(* CODESYS project CtaAppWagoModBus1.0.0.2.library
   Description: Modbus Library der CTA
      Mit WAGO unterstüzung.
   Version: 1.0.0.2
   Title: CtaAppWagoModbus
   Author: SIS
   Company: CTA
   Placeholder: CtaAppWagoModbus
   DocFormat: reStructuredText
   CompiledLibraryCompatibilityVersion: CODESYS V3.5 SP16 Patch 3
   LanguageModelAttribute: qualified-access-only
   DefaultNamespace: CtaAppWagoModbus

Project tree, tasks and I/O mapping:
  libraries: WagoAppPlcModbus, 1.1.4.8 (WAGO); Standard, 3.5.18.0 (System); CtaVisSymbols, 1.0.0.0 (CTA); CtaSysConfig, 1.0.0.0 (CTA); CtaAppTime, 1.0.0.0 (CTA); CtaAppBmk, 1.0.0.0 (CTA); VisuSymbols, 4.5.0.0 (System); VisuDialogs, * (System); CtaSysBase, 1.0.0.0 (CTA); CtaAppModbus, 1.0.0.0 (CTA)
  40 Visualizations/
    SERVER/
      visualisation VIS_ModBusServer
      INFO/
        visualisation VIS_ModBusAccesInfo
      PARAMETER/
        SERIAL/
          visualisation VIS_ModBusParameter_SERIAL
        TCP/
          visualisation VIS_ModBusParameter_TCP
        UDP/
          visualisation VIS_ModBusParameter_UDP
        visualisation VIS_ModBus_PopUp
    CLIENT/
      SERIAL Client/
        SERIAL PORT/
          visualisation VIS_ModBusSerialPort
          PARAMETER/
            SERIAL/
              visualisation VIS_ModBusParameter_Serial_Port_Control
            visualisation VIS_ModBus_PopUp_Serial_Port_Control
        SERIAL Client/
          visualisation VIS_ModBusSerialNode
          POPUP/
            PARAMETER/
              visualisation VIS_ModBusParameter_SERIAL_Client
            visualisation VIS_ModBus_Serial_NodePopUp
          visualisation VIS_ModBusSerialNode_QUERRY
        visualisation VIS_SERIAL_LINE_HORIZONTAL
        visualisation VIS_SERIAL_LINE_VERTIKAL
        visualisation VIS_MODBUS_SERIAL_LINE
      NETWORK Client/
        visualisation VIS_ModBusNetworkPortTcp
        TCP/
          visualisation VIS_ModBusTcpNode_QUERRY
          visualisation VIS_ModBusTcpNode
          POPUP/
            PARAMETER/
              visualisation VIS_ModBusParameter_TCP_Client
            visualisation VIS_ModBus_Tcpl_NodePopUp
        UDP/
        visualisation VIS_MODBUS_TCP_LINE
        visualisation VIS_TCP_LINE_HORIZONTAL
        visualisation VIS_TCP_LINE_VERTIKAL
      visualisation VIS_MODBUS_LINE
    HELPER/
      visualisation VIS_IP_INPUT
      visualisation VIS_IP_PARAMETER
      visualisation VIS_IP_PARAMETER_QUERRY
      visualisation VIS_IP_PARAMETER_BASE
    BMK/
      visualisation Node_BMK
      visualisation Node_BMK_QUERY
    DIALOG/
      visualisation ModBusPopUp
  30 Program Organization Units/
    JOB/
      function block fbJOB [ST]: metCheckToUnlinkUnlock, metCheckQuerryAdr, metLock, proAllJobsDone, metSetQuerry, metSetWriteWord, metGetResponse, metQuerryAyWordToAyWord, metQuerryAyBoolToAyWord, metResponsAyWordToAyBool, metResponsAyWordToAyWord, metCallAfterResponse, FB_INIT, metAnalytic, metMaxQuantity, metResetMissingLastAdr, metResetMissingFirstAdr
    CLIENT/
      NETWORK Client/
        TCP/
          function block fbMbTcpClient [ST]: actKeepAlive, FB_INIT, metCheckOnError, metFc4ReadInputRegister, actFC04, metFc2ReadDiscretInput, actFC15, metFc1ReadCoils, metFc3ReadHoldingRegister, metFc15WriteMultipleCoil, metFc16WriteHoldingRegisters, actFC01, actFC03, actConfig, actFC02, actFC16, proNodeReference, actFC43, sMajorMinorRevision, sProductCode, sVendorName, proModBusOK, metFc5WriteCoil, metFc6WriteHoldingRegister, actFC05, actFC06, proModBusErrorText, proModBusEnabled, proITF_BMK, metITF_BMK, actDelay
          function block fbMbTcpPortControll [ST]: metMbTcpClient, metSyncClient
        UDP/
          function block fbMbUdpClient [ST]: actFC16, metCheckOnError, actFcUserQuerry, metFc4ReadInputRegister, actFC04, actFC02, metFc2ReadDiscretInput, FB_INIT, metFc1ReadCoils, metFc15WriteMultipleCoil, metFc16WriteHoldingRegisters, actFC01, actFC03, actFC15, metFc3ReadHoldingRegister, actConfig, actFC43, sProductCode, sVendorName, sMajorMinorRevision, proModBusOK, metFc5WriteCoil, metFc6WriteHoldingRegister, actFC05, actFC06, proModBusErrorText, proModBusEnabled, metITF_BMK, proITF_BMK, actDelay
      SERIAL Client/
        function block fbMbSerialClient [ST]: actFC16, actFC15, actFC03, actFC01, metFc16WriteHoldingRegisters, metFc15WriteMultipleCoil, metFc3ReadHoldingRegister, metFc1ReadCoils, metCheckOnError, metFc2ReadDiscretInput, actFC02, actFC04, metFc4ReadInputRegister, FB_INIT, actConfig, proNodeReference, actFC43, sMajorMinorRevision, sProductCode, sVendorName, proModBusOK, actFC05, actFC06, metFc5WriteCoil, metFc6WriteHoldingRegister, proModBusErrorText, proModBusEnabled, metITF_BMK, proITF_BMK, actDelay
        function block fbMbSerialPortControll [ST]: metSyncClient, metMbSerialClient, actConfig
    SERVER/
      function block fbModBusServer [ST]: actConfig, actModBusServerTcp, actModBusServerUdp, actModBusServerSerial, metGetCoil, metSetDiscretInput, metGetHoldingRegister, metSetInputRegister, metAddSerialControll, metAddTcpControll, metAddUdpControll, metSetHoldingRegister, metSetCoil
      ACCES CONTROLL/
        function block fbAccesControll [ST]: beforeAccess, afterAccess, ALLOWBOOL
    CONVERTER/
      function fcWordBitToByte [ST]
      function fcCheckIp [ST]
      function fcSetInitialIPString [ST]
  00000000-0000-0000-0000-000000000000|D:\CoDeSys\LibrariesV3\trunk\Intern\CAA\CAA Template\3.4.0.0 draft\Placeholder.xml
  00000000-0000-0000-0000-000000000000|D:\CoDeSys\LibrariesV3\trunk\Intern\CAA\CAA Template\3.2.0.3 draft\Prefix.pdf
  00000000-0000-0000-0000-000000000000|D:\CoDeSys\LibrariesV3\trunk\Intern\CAA\CAA Template\3.5.2.0 draft\Placeholder.xml
  20 Structs/
    SERVER/
      PARAMETER/
        data type scModBusServerParameter
        TCP/
          data type scTcp
        UDP/
          data type scUdp
        SERIAL/
          data type scSerial
    CLIENT/
      SERIAL/
        data type scSerialPortParameter
        data type scSerialClientParameter
      NETWORK/
        data type scUdpClientParameter
        data type scTcpClientParameter
  50 Images/
  10 Documenation/
    global variables VersionHistory
    global variables readMe
  21 Interface/
    RTU/
      interface ITF_MbPortControllSerial: metMbSerialClient, metSyncClient
      interface ITF_SERIAL_NODE: proNodeReference
    ALL/
      interface ITF_MbClient: metFc16WriteHoldingRegisters, metFc15WriteMultipleCoil, metFc4ReadInputRegister, metFc3ReadHoldingRegister, metFc2ReadDiscretInput, metFc1ReadCoils, sProductCode, sVendorName, sMajorMinorRevision, proModBusOK, metFc5WriteCoil, metFc6WriteHoldingRegister, proModBusErrorText, proModBusEnabled, proITF_BMK, metITF_BMK
    NETWORK/
      interface ITF_TCP_NODE: proNodeReference
      interface ITF_UDP_NODE: proNodeReference
      interface ITF_MbPortControllTcp: metMbTcpClient, metSyncClient
    SERVER/
      interface ITF_SERVER: metAddSerialControll, metAddTcpControll, metAddUdpControll
  11 Library Parameter/
    global variables Parameter
  12 Konstanten/
  60 Textlisten/
    SERIAL/
      text list txtPhysikalLayer
      text list txtParity
      text list txtHandshake
      text list txtStopBits
  13 Globale Variablen/
    global variables GVL_CtaModBus
  text list GlobalTextList
*)

// 20 Structs/SERVER/PARAMETER/scModBusServerParameter
TYPE scModBusServerParameter :
    STRUCT
        scSerial    :   scSerial;
        scTcp       :   scTcp;
        scUdp       :   scUdp;
    END_STRUCT
END_TYPE

// 20 Structs/SERVER/PARAMETER/SERIAL/scSerial
TYPE scSerial :
    STRUCT
        fbxEnable           :   CtaSysConfig.fbBOOL;           // Serial Server Enable
        fbbyUnitId          :   CtaSysConfig.fbBYTE;           // Serial Server Id
        fbudiBaudrate       :   CtaSysConfig.fbUDINT;          // Serial Server Baudrate
        fbusiDataBits       :   CtaSysConfig.fbUSINT;          // Serial Server Databits 5..8
        fbiParity           :   CtaSysConfig.fbINT;            // WagoTypesCom.eTTYParity
        fbiStopBits         :   CtaSysConfig.fbINT;            // WagoTypesCom.eTTYStopBits
        fbiHandshake        :   CtaSysConfig.fbINT;            // WagoTypesCom.eTTYHandshake
        fbiPhysikal         :   CtaSysConfig.fbINT;            // WagoTypesCom.eTTYPhysicalLayer
        fbxRtuOrAscii       :   CtaSysConfig.fbBOOL;           // RTU = FALSE , ASCII = TRUE
        fbxEnableWatchDog   :   CtaSysConfig.fbBOOL;           // WatchDog Enable
        fbtWatchDog         :   CtaSysConfig.fbTIME;           // WatchDog Time
    END_STRUCT
END_TYPE

// 20 Structs/SERVER/PARAMETER/TCP/scTcp
TYPE scTcp :
    STRUCT
        fbxEnable           :   CtaSysConfig.fbBOOL;           // Tcp Server Enable    
        fbbyUnitId          :   CtaSysConfig.fbBYTE;           // Tcp Server Id
        fbwPort             :   CtaSysConfig.fbWORD;           // Tcp Server Port
        fbxKeepAlive        :   CtaSysConfig.fbBOOL;           // Tcp Server Keep Alive 
        fbtMaxIdleTime      :   CtaSysConfig.fbTIME;           // Tcp Server Max Offline Time
        fbtIntervall        :   CtaSysConfig.fbTIME;           // Tcp Server Intervall Time
        fbudiProbes         :   CtaSysConfig.fbUDINT;          // Tcp Server Retrys before give up 
        fbxEnableWatchDog   :   CtaSysConfig.fbBOOL;           // WatchDog Enable
        fbtWatchDog         :   CtaSysConfig.fbTIME;           // WatchDog Time
    END_STRUCT
END_TYPE

// 20 Structs/SERVER/PARAMETER/UDP/scUdp
TYPE scUdp :
    STRUCT
        fbxEnable       :   CtaSysConfig.fbBOOL;           // Udp Server Enable    
        fbbyUnitId      :   CtaSysConfig.fbBYTE;           // Udp Server Id
        fbwPort         :   CtaSysConfig.fbWORD;           // Udp Server Port  
        fbxEnableWatchDog   :   CtaSysConfig.fbBOOL;           // WatchDog Enable      
        fbtWatchDog     :   CtaSysConfig.fbTIME;           // WatchDog Time
    END_STRUCT
END_TYPE

// 20 Structs/CLIENT/NETWORK/scUdpClientParameter
TYPE scUdpClientParameter :
    STRUCT
        fbxEnable           :   CtaSysConfig.fbBOOL;           // Serial Server Enable        
        fbbyUnitId          :   CtaSysConfig.fbBYTE;           // Serial Server Id  
        fbstIp              :   CtaSysConfig.fbSTRING40;       // IP Adresse    
        fbwPort             :   CtaSysConfig.fbWORD;           // Port Nr          
        fbtTimeOut          :   CtaSysConfig.fbTIME;           // Timeout Time
        fbtScanRate         :   CtaSysConfig.fbTIME;           // Scan Rate Time
		fbtDelayRead		:	CtaSysConfig.fbTIME;		   // Read Delay
		fbtDelayWrite		:	CtaSysConfig.fbTIME;		   // Write Delay
    END_STRUCT
END_TYPE

// 20 Structs/CLIENT/SERIAL/scSerialPortParameter
TYPE scSerialPortParameter :
    STRUCT 
        fbudiBaudrate       :   CtaSysConfig.fbUDINT;          // Serial Server Baudrate
        fbusiDataBits       :   CtaSysConfig.fbUSINT;          // Serial Server Databits 5..8
        fbiParity           :   CtaSysConfig.fbINT;            // WagoTypesCom.eTTYParity
        fbiStopBits         :   CtaSysConfig.fbINT;            // WagoTypesCom.eTTYStopBits
        fbiHandshake        :   CtaSysConfig.fbINT;            // WagoTypesCom.eTTYHandshake
        fbiPhysikal         :   CtaSysConfig.fbINT;            // WagoTypesCom.eTTYPhysicalLayer
        fbxRtuOrAscii       :   CtaSysConfig.fbBOOL;           // RTU = FALSE , ASCII = TRUE
    END_STRUCT
END_TYPE

// 20 Structs/CLIENT/SERIAL/scSerialClientParameter
TYPE scSerialClientParameter :
    STRUCT
        fbxEnable           :   CtaSysConfig.fbBOOL;           // Serial Server Enable        
        fbbyUnitId          :   CtaSysConfig.fbBYTE;           // Serial Server Id        
        fbtTimeOut          :   CtaSysConfig.fbTIME;           // Timeout Time
        fbtScanRate         :   CtaSysConfig.fbTIME;           // Scan Rate Time
		fbtDelayRead		:	CtaSysConfig.fbTIME;		   // Read Delay
		fbtDelayWrite		:	CtaSysConfig.fbTIME;		   // Write Delay
    END_STRUCT
END_TYPE

// 20 Structs/CLIENT/NETWORK/scTcpClientParameter
TYPE scTcpClientParameter :
    STRUCT
        fbxEnable           :   CtaSysConfig.fbBOOL;           // Serial Server Enable       
        fbbyUnitId          :   CtaSysConfig.fbBYTE;           // Serial Server Id  
        fbstIp              :   CtaSysConfig.fbSTRING40;       // IP Adresse    
        fbwPort             :   CtaSysConfig.fbWORD;           // Port Nr          
        fbtTimeOut          :   CtaSysConfig.fbTIME;           // Timeout Time
        fbtScanRate         :   CtaSysConfig.fbTIME;           // Scan Rate Time
        fbxKeepAlive        :   CtaSysConfig.fbBOOL;           // Tcp Server Keep Alive 
        fbtMaxIdleTime      :   CtaSysConfig.fbTIME;           // Tcp Server Max Offline Time
        fbtIntervall        :   CtaSysConfig.fbTIME;           // Tcp Server Intervall Time
        fbudiProbes         :   CtaSysConfig.fbUDINT;          // Tcp Server Retrys before give up     
		fbtDelayRead		:	CtaSysConfig.fbTIME;		   // Read Delay
		fbtDelayWrite		:	CtaSysConfig.fbTIME;		   // Write Delay   
    END_STRUCT
END_TYPE

// 10 Documenation/VersionHistory
(* 

.. image:: ../../Images/CTA_Logo.jpg
   :align: right
   :width: 15% 

**Vorlage**   


============ =========== =========== ============================================
**Date**     **Version** **Author**  **Change**
------------ ----------- ----------- --------------------------------------------
04.03.2021   0.0.0.0     SIS         Vorlage erstellt

============ =========== =========== ============================================


*)
VAR_GLOBAL
    stInfo : STRING:= '0.0.0.0, Vorlage, CTA';
END_VAR

// 10 Documenation/readMe
(*

**ReadMe**
 
|	**Empfehlung**
|
|	Dokumentrieren Sie die Library für eine nachhaltige Entwicklung
|     
| *Beispiel* 
|
| Dies ist die Vorlage Library der CTA. Erstellen Sie ihre Library anhand dieser Vorlage.
*)

VAR_GLOBAL
    xReadMeDone              :   BOOL;
END_VAR

// 13 Globale Variablen/GVL_CtaModBus
{attribute 'qualified_only'}
VAR_GLOBAL   
    // {attribute 'hide'}
    byCountServer           : BYTE;     
    // {attribute 'hide'}     
    fbDeviceName            : WagoAppPlcModbus.FbIdentifyBaseObject:= ( _sVendorName            := Parameter.sVendorName,          
                                                                        _sProductCode           := Parameter.sProductCode,         
                                                                        _sMajorMinorRevision    := Parameter.sMajorMinorRevision);          
                                                      
END_VAR

// 11 Library Parameter/Parameter
{attribute 'qualified_only'}
VAR_GLOBAL CONSTANT
    sVendorName                 :   STRING(WagoAppPlcModbus.Parameter.MAX_IDENTIFICATION_MEMBER_LENGTH) := 'CTA AG';   
    sProductCode                :   STRING(WagoAppPlcModbus.Parameter.MAX_IDENTIFICATION_MEMBER_LENGTH) := 'CTA ModBus Device';
    sMajorMinorRevision         :   STRING(WagoAppPlcModbus.Parameter.MAX_IDENTIFICATION_MEMBER_LENGTH) := '1.0';    
    wQuantityReadTcpWord        :   WORD    :=  123;
    wQuantityReadTcpBool        :   WORD    := 1968;
    wQuantityReadSerialWord     :   WORD    :=  123;
    wQuantityReadSerialBool     :   WORD    := 1968;     
    wQuantityWriteTcpWord       :   WORD    :=  123;
    wQuantityWriteTcpBool       :   WORD    := 1968;
    wQuantityWriteSerialWord    :   WORD    :=   68;
    wQuantityWriteSerialBool    :   WORD    :=  123; 
END_VAR

// 30 Program Organization Units/CLIENT/SERIAL Client/fbMbSerialClient
FUNCTION_BLOCK fbMbSerialClient EXTENDS CtaSysBase.fbBASE IMPLEMENTS ITF_MbClient, ITF_SERIAL_NODE
VAR_INPUT
    ITF_MbPortControll          : ITF_MbPortControllSerial;   
END_VAR
VAR_OUTPUT
    xError                      : BOOL;
END_VAR
VAR
	ITF_BMK 					: CtaAppBmk.ITF_BMK;	
    xComAktive                  : BOOL;
    xDisabled                   : BOOL;
    byUnitId                    : BYTE;
    ITF_MbPortControllQuerry    : ITF_MbPortControllSerial; 
    xPortControllError          : BOOL;
    uiCountErrors               : UINT;    
    usiState                    : USINT := 1;
    fbTIMEFcs                   : CtaAppTime.fbTimeMeasurement;
    ltMessungFcs                : LTIME; 
    bIdOfCall                   : BYTE;
    TON_ScanRate                : TON;
    tonDelayRead				: Standard.TON;
	tonDelayWrite				: Standard.TON;
	xTrigDelayRead				: BOOL;
	xTrigDelayWrite				: BOOL; 
    xAllJobsDone                : BOOL;

    xErrorMbClientSerial        : BOOL;
    uiIdMbClientSerial          : UINT;
    
    
    (* FC1 *)
    fbJobFc1                    : fbJOB;
    xTrigFc1                    : BOOL;
    fbTIMEFc1                   : CtaAppTime.fbTimeMeasurement;
    ltMessungFc1                : LTIME;      
    (* FC2 *)
    fbJobFc2                    : fbJOB;
    xTrigFc2                    : BOOL; 
    fbTIMEFc2                   : CtaAppTime.fbTimeMeasurement;
    ltMessungFc2                : LTIME;      
    (* FC3 *)
    fbJobFc3                    : fbJOB;
    xTrigFc3                    : BOOL;      
    fbTIMEFc3                   : CtaAppTime.fbTimeMeasurement;
    ltMessungFc3                : LTIME;          
    (* FC4 *)
    fbJobFc4                    : fbJOB;
    xTrigFc4                    : BOOL;      
    fbTIMEFc4                   : CtaAppTime.fbTimeMeasurement;
    ltMessungFc4                : LTIME;      
    (* FC5 *)
    fbJobFc5                    : fbJOB;
    xTrigFc5                    : BOOL;      
    fbTIMEFc5                   : CtaAppTime.fbTimeMeasurement;
    ltMessungFc5                : LTIME;      
    (* FC6 *)
    fbJobFc6                    : fbJOB;
    xTrigFc6                    : BOOL;      
    fbTIMEFc6                   : CtaAppTime.fbTimeMeasurement;
    ltMessungFc6                : LTIME;      
    (* FC15 *)
    fbJobFc15                   : fbJOB;
    xTrigFc15                   : BOOL;   
    fbTIMEFc15                  : CtaAppTime.fbTimeMeasurement;
    ltMessungFc15               : LTIME;     
    (* FC16 *)   
    fbJobFc16                   : fbJOB;             
    xTrigFc16                   : BOOL;
    fbTIMEFc16                  : CtaAppTime.fbTimeMeasurement;
    ltMessungFc16               : LTIME;       
    (* FC43 *)   
    fbIdentifyObject			: WagoAppPlcModbus.FbIdentifyBaseObject;
	fbIdentifyMember3			: WagoAppPlcModbus.FbIdentifyMember_STRING(fbIdentifyObject,3);
	fbIdentifyMember4			: WagoAppPlcModbus.FbIdentifyMember_STRING(fbIdentifyObject,4);
	utIdentifyQuerry			: WagoAppPlcModbus.typMbQuery;
	utIdentifyResponse			: WagoAppPlcModbus.typMbResponse;           
    xTrigFc43                   : BOOL;
	xActiveFc43					: BOOL;
	xDoneFc43					: BOOL;
	tTimeOutFc43				: TIME;
    fbTIMEFc43                  : CtaAppTime.fbTimeMeasurement;
    ltMessungFc43               : LTIME;       	
    (* Parameter *)
    fbConfigFile                : CtaSysConfig.fbConfigFile;
    scParameter                 : scSerialClientParameter;    
END_VAR

(* Config File *)
actConfig();
(* Unit ID *)
byUnitId := scParameter.fbbyUnitId.byValue;
(* Is Enabled *)
IF scParameter.fbxEnable.xValue THEN
    (* Port Sync *)
    IF __QUERYINTERFACE(ITF_MbPortControll,ITF_MbPortControllQuerry) THEN
        xPortControllError := FALSE;  
        IF ITF_MbPortControllQuerry.metSyncClient(xAllJobsDone,bIdOfCall,THIS^) THEN
			(* Delay *)
			actDelay();
            (* FC1 *)
            actFC01();
            (* FC2 *)
            actFC02();
            (* FC3 *)
            actFC03();
            (* FC4 *)
            actFC04();
            (* FC5 *)
            actFC05();
            (* FC6 *)
            actFC06();
            (* FC15 *)
            actFC15();
            (* FC16 *)
            actFC16(); 
            (* FC43 *)
            actFC43(); 			
        END_IF;
    ELSE
        xPortControllError := TRUE;    
    END_IF;
    IF usiState >= 10 OR usiState = 0 THEN
        (* Check if all Jobs Done *)
        IF  fbJobFc1.xAllJobsDone  AND
            fbJobFc2.xAllJobsDone  AND
            fbJobFc3.xAllJobsDone  AND
            fbJobFc4.xAllJobsDone  AND
            fbJobFc5.xAllJobsDone  AND
            fbJobFc6.xAllJobsDone  AND			
            fbJobFc15.xAllJobsDone AND
            fbJobFc16.xAllJobsDone THEN
            (*Scan Rate *)
            TON_ScanRate(IN := NOT TON_ScanRate.Q,
                         PT := scParameter.fbtScanRate.tValue);
            xAllJobsDone := TRUE;             
            IF TON_ScanRate.Q THEN
                fbJobFc1.proAllJobsDone  := FALSE;
                fbJobFc2.proAllJobsDone  := FALSE;   
                fbJobFc3.proAllJobsDone  := FALSE;  
                fbJobFc4.proAllJobsDone  := FALSE;   
                fbJobFc5.proAllJobsDone  := FALSE;  
                fbJobFc6.proAllJobsDone  := FALSE; 	
                fbJobFc15.proAllJobsDone := FALSE;  
                fbJobFc16.proAllJobsDone := FALSE; 
                xAllJobsDone             := FALSE;    
                usiState := 1;
                (* Timer stopp *) 
                ltMessungFcs := fbTIMEFcs.stop();             
                (* Timer start *) 
                fbTIMEFcs.Start();      
            END_IF;        
        ELSE    
            usiState := 1;
        END_IF;   
    END_IF;
    
    xComAktive := fbJobFc1.wCountJobs  <> 0 OR 
                  fbJobFc2.wCountJobs  <> 0 OR
                  fbJobFc3.wCountJobs  <> 0 OR 
                  fbJobFc4.wCountJobs  <> 0 OR 
                  fbJobFc5.wCountJobs  <> 0 OR 
                  fbJobFc6.wCountJobs  <> 0 OR 				  
                  fbJobFc15.wCountJobs <> 0 OR
                  fbJobFc16.wCountJobs <> 0 ;  
                  
    (* Get Errors *)
    xError :=  fbJobFc1.eError <> WagoAppPlcModbus.eErrorModbus.OK OR 
               fbJobFc2.eError <> WagoAppPlcModbus.eErrorModbus.OK OR 
               fbJobFc3.eError <> WagoAppPlcModbus.eErrorModbus.OK OR 
               fbJobFc4.eError <> WagoAppPlcModbus.eErrorModbus.OK OR 
               fbJobFc5.eError <> WagoAppPlcModbus.eErrorModbus.OK OR 
               fbJobFc6.eError <> WagoAppPlcModbus.eErrorModbus.OK OR 			   
              fbJobFc15.eError <> WagoAppPlcModbus.eErrorModbus.OK OR 
              fbJobFc16.eError <> WagoAppPlcModbus.eErrorModbus.OK OR
              fbConfigFile.xError                                  OR
              xPortControllError;   
              
    IF NOT xError THEN
       uiCountErrors := 0;
    END_IF;
ELSE
    (* Reset States *)
    (* Port Sync *)
    IF __QUERYINTERFACE(ITF_MbPortControll,ITF_MbPortControllQuerry) THEN
        xPortControllError := FALSE;  
        xAllJobsDone       := FALSE;
        usiState           := 0;
        xError             := FALSE;
        xComAktive         := FALSE;
        xDisabled          := TRUE;
		xDoneFc43		   := FALSE;
        ITF_MbPortControllQuerry.metSyncClient(xDisabled,bIdOfCall,THIS^);
    END_IF; 
END_IF;

ACTION actFC16:
(* Trig FC16 *)
IF fbJobFc16.xIsLinked AND fbJobFc16.xIsQuerryReady AND NOT fbJobFc16.xIsLocked AND NOT fbJobFc16.xAllJobsDone AND tonDelayWrite.Q THEN
    fbJobFc16.metLock();
    xTrigFc16       := TRUE;
    fbTIMEFc16.Start();
ELSIF usiState = 8 AND (NOT fbJobFc16.xIsLinked OR fbJobFc16.xAllJobsDone) THEN
    usiState                    := usiState + 1; 
    fbJobFc16.proAllJobsDone    := TRUE;   
END_IF
(* Send Querry *)
IF usiState = 8 AND xTrigFc16 THEN
	xTrigDelayWrite := FALSE;
    ITF_MbPortControllQuerry.metMbSerialClient( tTimeOut    := scParameter.fbtTimeOut.tValue, 
                                                utQuery     := fbJobFc16.utQuery,
                                                xTrigger    := xTrigFc16,
                                                utResponse  := fbJobFc16.utResponse,
                                                xError      => xErrorMbClientSerial,
                                                uiID        => uiIdMbClientSerial);      
END_IF;
(* Get Response *) 
IF usiState = 8 AND NOT xTrigFc16 AND fbJobFc16.xIsLocked AND NOT fbJobFc16.xJobDone THEN    
    usiState            := usiState + 1;
    ltMessungFc16       := fbTIMEFc16.Stop();
    metCheckOnError(xErrorMbClientSerial);
    fbJobFc16.metCallAfterResponse(xErrorMbClientSerial,uiIdMbClientSerial);
END_IF;
END_ACTION

ACTION actFC15:
(* Trig FC15 *)
IF fbJobFc15.xIsLinked AND fbJobFc15.xIsQuerryReady AND NOT fbJobFc15.xIsLocked AND NOT fbJobFc15.xAllJobsDone AND tonDelayWrite.Q THEN
    fbJobFc15.metLock();
    xTrigFc15       := TRUE;
    fbTIMEFc15.Start();
ELSIF usiState = 7 AND (NOT fbJobFc15.xIsLinked OR fbJobFc15.xAllJobsDone) THEN
    usiState                    := usiState + 1; 
    fbJobFc15.proAllJobsDone    := TRUE;   
END_IF
(* Send Querry *)
IF usiState = 7 AND xTrigFc15 THEN
	xTrigDelayWrite := FALSE;
    ITF_MbPortControllQuerry.metMbSerialClient( tTimeOut    := scParameter.fbtTimeOut.tValue, 
                                                utQuery     := fbJobFc15.utQuery,
                                                xTrigger    := xTrigFc15,
                                                utResponse  := fbJobFc15.utResponse,
                                                xError      => xErrorMbClientSerial,
                                                uiID        => uiIdMbClientSerial); 
END_IF;
(* Get Response *) 
IF usiState = 7 AND NOT xTrigFc15 AND fbJobFc15.xIsLocked AND NOT fbJobFc15.xJobDone  THEN 
    usiState            := usiState + 1;
    ltMessungFc15       := fbTIMEFc15.Stop();
    metCheckOnError(xErrorMbClientSerial);
    fbJobFc15.metCallAfterResponse(xErrorMbClientSerial,uiIdMbClientSerial);
END_IF;
END_ACTION

ACTION actFC03:
(* Trig FC3 *)
IF fbJobFc3.xIsLinked AND fbJobFc3.xIsQuerryReady AND NOT fbJobFc3.xIsLocked AND NOT fbJobFc3.xAllJobsDone AND tonDelayRead.Q THEN
    fbJobFc3.metLock();
    xTrigFc3       := TRUE;
    fbTIMEFc3.Start();
ELSIF usiState = 3 AND (NOT fbJobFc3.xIsLinked OR fbJobFc3.xAllJobsDone) THEN
    usiState                := usiState + 1;
    fbJobFc3.proAllJobsDone := TRUE;    
END_IF
(* Send Querry *)
IF usiState = 3 AND xTrigFc3 THEN
	xTrigDelayRead 	:= FALSE;
    ITF_MbPortControllQuerry.metMbSerialClient( tTimeOut    := scParameter.fbtTimeOut.tValue, 
                                                utQuery     := fbJobFc3.utQuery,
                                                xTrigger    := xTrigFc3,
                                                utResponse  := fbJobFc3.utResponse,
                                                xError      => xErrorMbClientSerial,
                                                uiID        => uiIdMbClientSerial);       
END_IF;
(* Get Response *) 
IF usiState = 3 AND NOT xTrigFc3 AND fbJobFc3.xIsLocked AND NOT fbJobFc3.xJobDone  THEN
    usiState            := usiState + 1;
    ltMessungFc3        := fbTIMEFc3.Stop();
    metCheckOnError(xErrorMbClientSerial);
    fbJobFc3.metCallAfterResponse(xErrorMbClientSerial,uiIdMbClientSerial);
END_IF;
END_ACTION

ACTION actFC01:
(* Trig FC1 *)
IF fbJobFc1.xIsLinked AND fbJobFc1.xIsQuerryReady AND NOT fbJobFc1.xIsLocked AND NOT fbJobFc1.xAllJobsDone AND tonDelayRead.Q THEN
    fbJobFc1.metLock();
    xTrigFc1       := TRUE;
    fbTIMEFc1.Start();
ELSIF usiState = 1 AND (NOT fbJobFc1.xIsLinked OR fbJobFc1.xAllJobsDone) THEN
    usiState                := usiState + 1;    
    fbJobFc1.proAllJobsDone := TRUE;
END_IF
(* Send Querry *)
IF usiState = 1 AND xTrigFc1 THEN
	xTrigDelayRead 	:= FALSE;
    ITF_MbPortControllQuerry.metMbSerialClient( tTimeOut    := scParameter.fbtTimeOut.tValue, 
                                                utQuery     := fbJobFc1.utQuery,
                                                xTrigger    := xTrigFc1,
                                                utResponse  := fbJobFc1.utResponse,
                                                xError      => xErrorMbClientSerial,
                                                uiID        => uiIdMbClientSerial);     
END_IF;
(* Get Response *) 
IF usiState = 1 AND NOT xTrigFc1 AND fbJobFc1.xIsLocked AND NOT fbJobFc1.xJobDone  THEN      
    usiState            := usiState + 1;
    ltMessungFc1        := fbTIMEFc1.Stop();
    metCheckOnError(xErrorMbClientSerial);
    fbJobFc1.metCallAfterResponse(xErrorMbClientSerial,uiIdMbClientSerial);
END_IF;
END_ACTION

METHOD FINAL metFc16WriteHoldingRegisters
VAR_INPUT
    wADR                :   WORD;
    pWord               :   POINTER TO WORD;
    uiQuantity          :   UINT;               // Anzahl Words Max 125
    wOffset             :   WORD;               // Pointer Offset wenn Array > 125 WORD    
END_VAR
VAR
    diCurrentJop        :   DINT;
    uiFor               :   UINT;
END_VAR
(* Limit Write Holding Registers *)
uiQuantity := LIMIT(1,uiQuantity,125);
(* Check if valid Pointer and Adress *)
IF pWord <> 0 AND wOffset + uiQuantity <= 16#FFFF + 1 AND wADR <= 16#FFFF THEN
    (* Link Adress *)
    fbJobFc16.bUnitId       := byUnitId;
    fbJobFc16.bFunctionCode := 16;
    fbJobFc16.bFunctionCode := 16;
    fbJobFc16.xIsBoolQuerry := FALSE;
    fbJobFc16.xIsSerialJob  := TRUE;        
    fbJobFc16.metCheckQuerryAdr(wADR,uiQuantity,pWord,wOffset);
END_IF;
END_METHOD

METHOD FINAL metFc15WriteMultipleCoil
VAR_INPUT
    wADR                :   WORD;
    pByte               :   POINTER TO BYTE;
    uiQuantity          :   UINT;               // Anzahl Coils Max 2000   
    wOffset             :   WORD;               // Pointer Offset wenn BOOL Array > 125     
END_VAR
VAR
    diCurrentJop        :   DINT;
    uiFor               :   UINT;
    usiCountWords       :   UINT;
    wTempValue          :   WORD;    
END_VAR
(* Limit Write Multiple Coil *)
uiQuantity := LIMIT(1,uiQuantity,2000);
(* Check if valid Pointer and Adress *)
IF pByte <> 0 AND wOffset + uiQuantity <= 16#FFFF + 1 AND wADR <= 16#FFFF THEN
    (* Link Adress *)
    fbJobFc15.bUnitId       := byUnitId;
    fbJobFc15.bFunctionCode := 15;
    fbJobFc15.xIsBoolQuerry := TRUE;
    fbJobFc15.xIsSerialJob  := TRUE;           
    fbJobFc15.metCheckQuerryAdr(wADR,uiQuantity,pByte,wOffset);    
END_IF;
END_METHOD

METHOD FINAL metFc3ReadHoldingRegister
VAR_INPUT
    wADR                :   WORD;
    pWord               :   POINTER TO WORD;
    uiQuantity          :   UINT;               // Anzahl Words Max 125
    wOffset             :   WORD;               // Pointer Offset wenn WORD Array > 125    
END_VAR
VAR
    diCurrentJop        :   DINT;
    uiFor               :   UINT;
    pBaseAdr            :   POINTER TO WORD;
END_VAR
(* Limit Holding Register *)
uiQuantity := LIMIT(1,uiQuantity,125);
(* Check if valid Pointer and Adress *)
IF pWord <> 0 AND wOffset + uiQuantity <= 16#FFFF + 1 AND wADR <= 16#FFFF THEN
    (* Link Adress *)
    fbJobFc3.bUnitId       := byUnitId;
    fbJobFc3.bFunctionCode := 3;
    fbJobFc3.xIsBoolQuerry := FALSE;
    fbJobFc3.xIsSerialJob  := TRUE;       
    fbJobFc3.metCheckQuerryAdr(wADR,uiQuantity,pWord,wOffset);     
END_IF;
END_METHOD

METHOD FINAL metFc1ReadCoils
VAR_INPUT
    wADR                :   WORD;
    pByte               :   POINTER TO BYTE;
    uiQuantity          :   UINT;               // Anzahl Coils Max 2000
    wOffset             :   WORD;               // Pointer Offset wenn BOOL Array > 125     
END_VAR
VAR
    diCurrentJop        :   DINT;
    uiFor               :   UINT;
    usiCountWords       :   UINT;
    wTempValue          :   WORD;
END_VAR
(* Limit Coils *)
uiQuantity := LIMIT(1,uiQuantity,2000);
(* Check if valid Pointer and Adress *)
IF pByte <> 0 AND wOffset + uiQuantity <= 16#FFFF + 1 AND wADR <= 16#FFFF THEN
    (* Link Adress *)
    fbJobFc1.bUnitId       := byUnitId;
    fbJobFc1.bFunctionCode := 1;
    fbJobFc1.xIsBoolQuerry := TRUE;
    fbJobFc1.xIsSerialJob  := TRUE;        
    fbJobFc1.metCheckQuerryAdr(wADR,uiQuantity,pByte,wOffset);        
END_IF;
END_METHOD

METHOD PRIVATE FINAL metCheckOnError : BOOL
VAR_INPUT
    xError  :  BOOL;
END_VAR
IF xError THEN
    uiCountErrors  := uiCountErrors + 1;
    metCheckOnError := TRUE;
END_IF
END_METHOD

METHOD FINAL metFc2ReadDiscretInput
VAR_INPUT
    wADR                :   WORD;
    pByte               :   POINTER TO BYTE;
    uiQuantity          :   UINT;               // Anzahl BOOL Max 2000
    wOffset             :   WORD;               // Pointer Offset wenn BOOL Array > 125    
END_VAR
VAR
    diCurrentJop        :   DINT;
    uiFor               :   UINT;
    usiCountWords       :   UINT;    
    wTempValue          :   WORD;
    pBaseAdr            :   POINTER TO BYTE;
END_VAR
(* Limit Discret Inputs *)
uiQuantity := LIMIT(1,uiQuantity,2000);
(* Check if valid Pointer and Adress *)
IF pByte <> 0 AND wOffset + uiQuantity <= 16#FFFF + 1 AND wADR <= 16#FFFF THEN
    (* Link Adress *)
    fbJobFc2.bUnitId       := byUnitId;
    fbJobFc2.bFunctionCode := 2;
    fbJobFc2.xIsBoolQuerry := TRUE;
    fbJobFc2.xIsSerialJob  := TRUE;        
    fbJobFc2.metCheckQuerryAdr(wADR,uiQuantity,pByte,wOffset);    
END_IF;
END_METHOD

ACTION actFC02:
(* Trig FC2 *)
IF fbJobFc2.xIsLinked AND fbJobFc2.xIsQuerryReady AND NOT fbJobFc2.xIsLocked AND NOT fbJobFc2.xAllJobsDone AND tonDelayRead.Q THEN
    fbJobFc2.metLock();
    xTrigFc2       := TRUE;
    fbTIMEFc2.Start();
ELSIF usiState = 2 AND (NOT fbJobFc2.xIsLinked OR fbJobFc2.xAllJobsDone) THEN
    usiState                := usiState + 1; 
    fbJobFc2.proAllJobsDone := TRUE;   
END_IF
(* Send Querry *)
IF usiState = 2 AND xTrigFc2 THEN
	xTrigDelayRead 	:= FALSE;
    ITF_MbPortControllQuerry.metMbSerialClient( tTimeOut    := scParameter.fbtTimeOut.tValue, 
                                                utQuery     := fbJobFc2.utQuery,
                                                xTrigger    := xTrigFc2,
                                                utResponse  := fbJobFc2.utResponse,
                                                xError      => xErrorMbClientSerial,
                                                uiID        => uiIdMbClientSerial);   
END_IF;
(* Get Response *) 
IF usiState = 2 AND NOT xTrigFc2 AND fbJobFc2.xIsLocked AND NOT fbJobFc2.xJobDone  THEN
    usiState            := usiState + 1;
    ltMessungFc2        := fbTIMEFc2.Stop();
    metCheckOnError(xErrorMbClientSerial);
    fbJobFc2.metCallAfterResponse(xErrorMbClientSerial,uiIdMbClientSerial);
END_IF;
END_ACTION

ACTION actFC04:
(* Trig FC4 *)
IF fbJobFc4.xIsLinked AND fbJobFc4.xIsQuerryReady AND NOT fbJobFc4.xIsLocked AND NOT fbJobFc4.xAllJobsDone AND tonDelayRead.Q THEN
    fbJobFc4.metLock();
    xTrigFc4       := TRUE;
    fbTIMEFc4.Start();
ELSIF usiState = 4 AND (NOT fbJobFc4.xIsLinked OR fbJobFc4.xAllJobsDone)  THEN
    usiState                := usiState + 1; 
    fbJobFc4.proAllJobsDone := TRUE;   
END_IF
(* Send Querry *)
IF usiState = 4 AND xTrigFc4 THEN
	xTrigDelayRead 	:= FALSE;
    ITF_MbPortControllQuerry.metMbSerialClient( tTimeOut    := scParameter.fbtTimeOut.tValue, 
                                                utQuery     := fbJobFc4.utQuery,
                                                xTrigger    := xTrigFc4,
                                                utResponse  := fbJobFc4.utResponse,
                                                xError      => xErrorMbClientSerial,
                                                uiID        => uiIdMbClientSerial);          
END_IF;
(* Get Response *) 
IF usiState = 4 AND NOT xTrigFc4 AND fbJobFc4.xIsLocked AND NOT fbJobFc4.xJobDone  THEN
    usiState            := usiState + 1;
    ltMessungFc4        := fbTIMEFc4.Stop();
    metCheckOnError(xErrorMbClientSerial);
    fbJobFc4.metCallAfterResponse(xErrorMbClientSerial,uiIdMbClientSerial);
END_IF;
END_ACTION

METHOD FINAL metFc4ReadInputRegister
VAR_INPUT
    wADR                :   WORD;
    pWord               :   POINTER TO WORD;
    uiQuantity          :   UINT;               // Anzahl Words Max 125
    wOffset             :   WORD;               // Pointer Offset wenn WORD Array > 125   
END_VAR
VAR
    diCurrentJop        :   DINT;
    uiFor               :   UINT;
    pBaseAdr            :   POINTER TO WORD;
END_VAR
(* Limit Read Input Register *)
uiQuantity := LIMIT(1,uiQuantity,125);
(* Check if valid Pointer and Adress *)
IF pWord <> 0 AND wOffset + uiQuantity <= 16#FFFF + 1 AND wADR <= 16#FFFF THEN
    (* Link Adress *)
    fbJobFc4.bUnitId       := byUnitId;
    fbJobFc4.bFunctionCode := 4;
    fbJobFc4.xIsBoolQuerry := FALSE;
    fbJobFc4.xIsSerialJob  := TRUE;        
    fbJobFc4.metCheckQuerryAdr(wADR,uiQuantity,pWord,wOffset);        
END_IF;
END_METHOD

//FB_Init ist immer implizit verfügbar und wird primär für die Initialisierung verwendet.
//Der Rückgabewert wird nicht ausgewertet. Für gezielte Einflussnahme können Sie
//die Methoden explizit deklarieren und darin mit dem Standard-Initialisierungscode 
//zusätzlichen Code bereitstellen. Sie können den Rückgabewert auswerten.
METHOD FB_Init: BOOL
VAR_INPUT    
bInitRetains: BOOL; // TRUE: Die Retain-Variablen werden initialisiert (Reset warm / Reset kalt)    
bInCopyCode: BOOL;  // TRUE: Die Instanz wird danach in den Kopiercode kopiert (Online-Change)
END_VAR
xTrigFc1    := FALSE;
xTrigFc2    := FALSE;
xTrigFc3    := FALSE;
xTrigFc4    := FALSE;
xTrigFc15   := FALSE;
xTrigFc16   := FALSE;
usiState    := 0;
END_METHOD

ACTION actConfig:
(* Config File *)
fbConfigFile();

scParameter.fbxEnable           (_usiParaNr :=  1, itfConfigFb := fbconfigFile                                           );
scparameter.fbbyUnitId          (_usiParaNr :=  2, itfConfigFb := fbconfigFile , _MinInit := 0      ,_MaxInit := 247     );
scparameter.fbtTimeOut          (_usiParaNr :=  3, itfConfigFb := fbconfigFile , _MinInit := T#50MS ,_MaxInit := T#10M   );
scparameter.fbtScanRate         (_usiParaNr :=  4, itfConfigFb := fbconfigFile , _MinInit := T#00MS ,_MaxInit := T#10M   );
scParameter.fbtDelayRead		(_usiParaNr :=  5, itfConfigFb := fbconfigFile , _MinInit := T#1MS  ,_MaxInit := T#10M   );	
scParameter.fbtDelayWrite		(_usiParaNr :=  6, itfConfigFb := fbconfigFile , _MinInit := T#1MS  ,_MaxInit := T#10M   );
END_ACTION

PROPERTY proNodeReference : REFERENCE TO fbMbSerialClient
GET
proNodeReference REF= THIS^;
END_GET
END_PROPERTY

ACTION actFC43:
(* Trig FC43 *)
IF usiState = 9 AND NOT xDoneFc43 AND NOT xActiveFc43 THEN
	xTrigFc43       	:= TRUE;
	xActiveFc43			:= TRUE;
	tTimeOutFc43		:= T#1S;
	utIdentifyQuerry.bUnitId			:= byUnitId;
	utIdentifyQuerry.bFunctionCode		:= 43;	
	utIdentifyQuerry.IIdentifyObject	:= fbIdentifyObject;	
    fbTIMEFc43.Start();
ELSIF usiState = 9 AND NOT xActiveFc43 THEN
    usiState                := usiState + 1; 
END_IF
(* Send Querry *)
IF usiState = 9 AND xTrigFc43 THEN
    ITF_MbPortControllQuerry.metMbSerialClient( tTimeOut    := tTimeOutFc43, 
                                                utQuery     := utIdentifyQuerry,
                                                xTrigger    := xTrigFc43,
                                                utResponse  := utIdentifyResponse,
                                                xError      => xErrorMbClientSerial,
                                                uiID        => uiIdMbClientSerial);          
END_IF;
(* Get Response *) 
IF usiState = 9 ANd NOT xTrigFc43 AND xActiveFc43 AND NOT xDoneFc43 THEN
    usiState            := usiState + 1;
    ltMessungFc43       := fbTIMEFc43.Stop();
	xActiveFc43 		:= FALSE;
	IF uiIdMbClientSerial = 16#99 THEN
		xDoneFc43			:= FALSE;
	ELSE
		xDoneFc43			:= TRUE;
	END_IF;
END_IF;
END_ACTION

{attribute 'monitoring' := 'call'}
PROPERTY sMajorMinorRevision : STRING(WagoAppPlcModbus.Parameter.MAX_IDENTIFICATION_MEMBER_LENGTH)
GET
sMajorMinorRevision := fbIdentifyObject.sMajorMinorRevision;
END_GET
END_PROPERTY

{attribute 'monitoring' := 'call'}
PROPERTY sProductCode : STRING(WagoAppPlcModbus.Parameter.MAX_IDENTIFICATION_MEMBER_LENGTH)
GET
sProductCode := fbIdentifyObject.sProductCode;
END_GET
END_PROPERTY

{attribute 'monitoring' := 'call'}
PROPERTY sVendorName : STRING(WagoAppPlcModbus.Parameter.MAX_IDENTIFICATION_MEMBER_LENGTH)
GET
sVendorName := fbIdentifyObject.sVendorName;
END_GET
END_PROPERTY

PROPERTY proModBusOK : BOOL
GET
proModBusOK := xComAktive AND NOT xError;
END_GET
END_PROPERTY

ACTION actFC05:
(* Trig FC15 *)
IF fbJobFc5.xIsLinked AND fbJobFc5.xIsQuerryReady AND NOT fbJobFc5.xIsLocked AND NOT fbJobFc5.xAllJobsDone AND tonDelayWrite.Q THEN
    fbJobFc5.metLock();
    xTrigFc5       := TRUE;
    fbTIMEFc5.Start();
ELSIF usiState = 5 AND (NOT fbJobFc5.xIsLinked OR fbJobFc5.xAllJobsDone) THEN
    usiState                    := usiState + 1; 
    fbJobFc5.proAllJobsDone    := TRUE;   
END_IF
(* Send Querry *)
IF usiState = 5 AND xTrigFc5 THEN
	xTrigDelayWrite := FALSE;
    ITF_MbPortControllQuerry.metMbSerialClient( tTimeOut    := scParameter.fbtTimeOut.tValue, 
                                                utQuery     := fbJobFc5.utQuery,
                                                xTrigger    := xTrigFc5,
                                                utResponse  := fbJobFc5.utResponse,
                                                xError      => xErrorMbClientSerial,
                                                uiID        => uiIdMbClientSerial); 
END_IF;
(* Get Response *) 
IF usiState = 5 AND NOT xTrigFc5 AND fbJobFc5.xIsLocked AND NOT fbJobFc5.xJobDone  THEN 
    usiState            := usiState + 1;
    ltMessungFc5       := fbTIMEFc5.Stop();
    metCheckOnError(xErrorMbClientSerial);
    fbJobFc5.metCallAfterResponse(xErrorMbClientSerial,uiIdMbClientSerial);
END_IF;
END_ACTION

ACTION actFC06:
(* Trig FC6 *)
IF fbJobFc6.xIsLinked AND fbJobFc6.xIsQuerryReady AND NOT fbJobFc6.xIsLocked AND NOT fbJobFc6.xAllJobsDone AND tonDelayWrite.Q THEN
    fbJobFc6.metLock();
    xTrigFc6       := TRUE;
    fbTIMEFc6.Start();
ELSIF usiState = 6 AND (NOT fbJobFc6.xIsLinked OR fbJobFc6.xAllJobsDone) THEN
    usiState                    := usiState + 1; 
    fbJobFc6.proAllJobsDone    := TRUE;   
END_IF
(* Send Querry *)
IF usiState = 6 AND xTrigFc6 THEN
	xTrigDelayWrite := FALSE;
    ITF_MbPortControllQuerry.metMbSerialClient( tTimeOut    := scParameter.fbtTimeOut.tValue, 
                                                utQuery     := fbJobFc6.utQuery,
                                                xTrigger    := xTrigFc6,
                                                utResponse  := fbJobFc6.utResponse,
                                                xError      => xErrorMbClientSerial,
                                                uiID        => uiIdMbClientSerial);      
END_IF;
(* Get Response *) 
IF usiState = 6 AND NOT xTrigFc6 AND fbJobFc6.xIsLocked AND NOT fbJobFc6.xJobDone THEN    
    usiState            := usiState + 1;
    ltMessungFc6        := fbTIMEFc6.Stop();
    metCheckOnError(xErrorMbClientSerial);
    fbJobFc6.metCallAfterResponse(xErrorMbClientSerial,uiIdMbClientSerial);
END_IF;
END_ACTION

METHOD FINAL metFc5WriteCoil
VAR_INPUT
    wADR                :   WORD;
    pByte               :   POINTER TO BYTE;
    uiQuantity          :   UINT;               // Anzahl Coils Max 2000   
    wOffset             :   WORD;               // Pointer Offset wenn BOOL Array > 125     
END_VAR
VAR
    diCurrentJop        :   DINT;
    uiFor               :   UINT;
    usiCountWords       :   UINT;
    wTempValue          :   WORD;    
END_VAR
(* Limit Write Multiple Coil *)
uiQuantity := LIMIT(1,uiQuantity,1);
(* Check if valid Pointer and Adress *)
IF pByte <> 0 AND wOffset + uiQuantity <= 16#FFFF + 1 AND wADR <= 16#FFFF THEN
    (* Link Adress *)
    fbJobFc5.bUnitId       := byUnitId;
    fbJobFc5.bFunctionCode := 5;
    fbJobFc5.xIsBoolQuerry := TRUE;
    fbJobFc5.xIsSerialJob  := TRUE;           
    fbJobFc5.metCheckQuerryAdr(wADR,uiQuantity,pByte,wOffset);    
END_IF;
END_METHOD

METHOD FINAL metFc6WriteHoldingRegister
VAR_INPUT
    wADR                :   WORD;
    pWord               :   POINTER TO WORD;
    uiQuantity          :   UINT;               // Anzahl Words Max 125
    wOffset             :   WORD;               // Pointer Offset wenn Array > 125 WORD    
END_VAR
VAR
    diCurrentJop        :   DINT;
    uiFor               :   UINT;
END_VAR
(* Limit Write Holding Registers *)
uiQuantity := LIMIT(1,uiQuantity,1);
(* Check if valid Pointer and Adress *)
IF pWord <> 0 AND wOffset + uiQuantity <= 16#FFFF + 1 AND wADR <= 16#FFFF THEN
    (* Link Adress *)
    fbJobFc6.bUnitId       := byUnitId;
    fbJobFc6.bFunctionCode := 6;
    fbJobFc6.xIsBoolQuerry := FALSE;
    fbJobFc6.xIsSerialJob  := TRUE;        
    fbJobFc6.metCheckQuerryAdr(wADR,uiQuantity,pWord,wOffset);
END_IF;
END_METHOD

PROPERTY proModBusErrorText : String(20)
GET
proModBusErrorText := TO_STRING(MAX(fbJobFc1.eError,fbJobFc2.eError,fbJobFc3.eError,fbJobFc4.eError,fbJobFc5.eError,fbJobFc6.eError,fbJobFc15.eError,fbJobFc16.eError));
END_GET
END_PROPERTY

PROPERTY proModBusEnabled : BOOL
GET
proModBusEnabled := scParameter.fbxEnable.xValue;
END_GET
END_PROPERTY

METHOD metITF_BMK
VAR_INPUT
	ITF_BMK_IN : CtaAppBmk.ITF_BMK;
END_VAR
ITF_BMK := ITF_BMK_IN;
END_METHOD

PROPERTY proITF_BMK : CtaAppBmk.ITF_BMK
GET
proITF_BMK := ITF_BMK;
END_GET
END_PROPERTY

ACTION actDelay:
(* Delay Read *)
tonDelayRead(	IN	:= xTrigDelayRead AND xTrigDelayWrite,
			 	PT 	:= scParameter.fbtDelayRead.proValue);
(* Delay Write *)
tonDelayWrite(	IN	:= xTrigDelayRead AND xTrigDelayWrite,
			 	PT 	:= scParameter.fbtDelayWrite.proValue);
				
(* Trig *)
xTrigDelayRead 	:= TRUE;
xTrigDelayWrite := TRUE;
END_ACTION

END_FUNCTION_BLOCK

// 21 Interface/ALL/ITF_MbClient
INTERFACE ITF_MbClient EXTENDS CtaSysBase.ITF_BASE

METHOD metFc16WriteHoldingRegisters
VAR_INPUT
    wADR                :   WORD;
    pWord               :   POINTER TO WORD;
    uiQuantity          :   UINT;               // Anzahl Words Max 125
    wOffset             :   WORD;               // Pointer Offset wenn Array > 125 WORD    
END_VAR
END_METHOD

METHOD metFc15WriteMultipleCoil
VAR_INPUT
    wADR                :   WORD;
    pByte               :   POINTER TO BYTE;
    uiQuantity          :   UINT;               // Anzahl Coils Max 2000   
    wOffset             :   WORD;               // Pointer Offset wenn BOOL Array > 125     
END_VAR
END_METHOD

METHOD metFc4ReadInputRegister
VAR_INPUT
    wADR                :   WORD;
    pWord               :   POINTER TO WORD;
    uiQuantity          :   UINT;               // Anzahl Words Max 125
    wOffset             :   WORD;               // Pointer Offset wenn WORD Array > 125   
END_VAR
END_METHOD

METHOD metFc3ReadHoldingRegister
VAR_INPUT
    wADR                :   WORD;
    pWord               :   POINTER TO WORD;
    uiQuantity          :   UINT;               // Anzahl Words Max 125
    wOffset             :   WORD;               // Pointer Offset wenn WORD Array > 125    
END_VAR
END_METHOD

METHOD metFc2ReadDiscretInput
VAR_INPUT
    wADR                :   WORD;
    pByte               :   POINTER TO BYTE;
    uiQuantity          :   UINT;               // Anzahl BOOL Max 2000
    wOffset             :   WORD;               // Pointer Offset wenn BOOL Array > 125    
END_VAR
END_METHOD

METHOD metFc1ReadCoils
VAR_INPUT
    wADR                :   WORD;
    pByte               :   POINTER TO BYTE;
    uiQuantity          :   UINT;               // Anzahl Coils Max 2000
    wOffset             :   WORD;               // Pointer Offset wenn BOOL Array > 125     
END_VAR
END_METHOD

{attribute 'monitoring' := 'call'}
PROPERTY sProductCode : STRING(WagoAppPlcModbus.Parameter.MAX_IDENTIFICATION_MEMBER_LENGTH)
GET
END_GET
END_PROPERTY

{attribute 'monitoring' := 'call'}
PROPERTY sVendorName : STRING(WagoAppPlcModbus.Parameter.MAX_IDENTIFICATION_MEMBER_LENGTH)
GET
END_GET
END_PROPERTY

{attribute 'monitoring' := 'call'}
PROPERTY sMajorMinorRevision : STRING(WagoAppPlcModbus.Parameter.MAX_IDENTIFICATION_MEMBER_LENGTH)
GET
END_GET
END_PROPERTY

PROPERTY proModBusOK : BOOL
GET
END_GET
END_PROPERTY

METHOD FINAL metFc5WriteCoil
VAR_INPUT
    wADR                :   WORD;
    pByte               :   POINTER TO BYTE;
    uiQuantity          :   UINT;               // Anzahl Coils Max 2000   
    wOffset             :   WORD;               // Pointer Offset wenn BOOL Array > 125     
END_VAR
END_METHOD

METHOD FINAL metFc6WriteHoldingRegister
VAR_INPUT
    wADR                :   WORD;
    pWord               :   POINTER TO WORD;
    uiQuantity          :   UINT;               // Anzahl Words Max 125
    wOffset             :   WORD;               // Pointer Offset wenn Array > 125 WORD    
END_VAR
END_METHOD

PROPERTY proModBusErrorText : String(20)
GET
END_GET
END_PROPERTY

PROPERTY proModBusEnabled : BOOL
GET
END_GET
END_PROPERTY

PROPERTY proITF_BMK : CtaAppBmk.ITF_BMK
GET
END_GET
END_PROPERTY

METHOD metITF_BMK
VAR_INPUT
	ITF_BMK_IN : CtaAppBmk.ITF_BMK;
END_VAR
END_METHOD

END_INTERFACE

// 21 Interface/RTU/ITF_SERIAL_NODE
INTERFACE ITF_SERIAL_NODE EXTENDS __SYSTEM.IQueryInterface

PROPERTY proNodeReference : REFERENCE TO fbMbSerialClient
GET
END_GET
END_PROPERTY

END_INTERFACE

// 21 Interface/RTU/ITF_MbPortControllSerial
INTERFACE ITF_MbPortControllSerial EXTENDS __SYSTEM.IQueryInterface

METHOD metMbSerialClient
VAR_IN_OUT
    tTimeOut     :  TIME;  
    utQuery      :  WagoAppPlcModbus.typMbQuery;
    xTrigger     :  BOOL;
    utResponse   :  WagoAppPlcModbus.typMbResponse;
END_VAR
VAR_OUTPUT
    xError       :  BOOL;
    uiID         :  UINT;
END_VAR
END_METHOD

METHOD metSyncClient : BOOL
VAR_IN_OUT
    xAllJobsDone    : BOOL;
    bIdOfCall       : BYTE;
END_VAR
VAR_INPUT
    ITF_SERIAL_NODE : ITF_SERIAL_NODE;
END_VAR
END_METHOD

END_INTERFACE

// 30 Program Organization Units/JOB/fbJOB
FUNCTION_BLOCK fbJOB
VAR_INPUT
    bUnitId                 :   BYTE;
    bFunctionCode           :   BYTE;
    utResponse              :   typMbResponse;  
    xIsSerialJob            :   BOOL;     
    xIsBoolQuerry           :   BOOL;                  // TRUE = Bool Querry    
END_VAR                     
VAR_OUTPUT                
    wStartAdress            :   WORD;
    wStopAdress             :   WORD;  
    uiQuantity              :   UINT;  
    utQuery                 :   typMbQuery  := (IIdentifyObject := GVL_CtaModBus.fbDeviceName);     
    eError                  :   WagoAppPlcModbus.eErrorModbus; 
    diErrorAdress           :   DINT := -1;                                  
END_VAR                     
VAR     
    eErrorCurrent           :   WagoAppPlcModbus.eErrorModbus;   
    wMaxQuantity            :   WORD;
    xFirstRequestDone       :   BOOL;            
    xIsLinked               :   BOOL;
    xIsLocked               :   BOOL;
    xIsQuerryReady          :   BOOL;
    xJobDone                :   BOOL;
    xDataAvailable          :   BOOL;
    xAllJobsDone            :   BOOL;
    diSandwichAdress        :   DINT    := -1;
    wCountJobs              :   DINT;
    wCountJobsTemp          :   DINT;
    diFirstDetectetAdress   :   DINT    := -1;
    diLastDetectetAdress    :   DINT    := -1;
    diTempDetectetAdress    :   DINT    := -1;
    fbTIME                  :   CtaAppTime.fbTimeMeasurement;
    ltMessung               :   LTIME;      
	fbTimeDiscareJob		:	CtaAppTime.fbTimeMeasurement;
	xCheckLastAdr			:	BOOL;
	xCheckFirstAdr			:	BOOL;
END_VAR

METHOD PRIVATE metCheckToUnlinkUnlock : BOOL
VAR_INPUT
    wAdressIn        :   WORD;
    uiQuantityIn     :   UINT; 
END_VAR
VAR
    diFor            :  DINT;
END_VAR
IF xJobDone THEN
    IF (wAdressIn + uiQuantityIn - 1 = wStopAdress AND xIsLocked) OR fbTimeDiscareJob.Stop() > LTIME#30S THEN 
		IF fbTimeDiscareJob.Stop() > LTIME#30S THEN
			xIsLinked               := FALSE;   
			xIsLocked               := FALSE;   
			xJobDone                := FALSE;   
			xAllJobsDone            := FALSE; 
			xFirstRequestDone		:= FALSE; 
			diSandwichAdress        := -1;
			diErrorAdress           := -1;
			eError                  :=  0;
			eErrorCurrent           :=  0;
			wCountJobs              :=  0;
			wCountJobsTemp          :=  0;
			diFirstDetectetAdress   := -1;
			diLastDetectetAdress    := -1;
			diTempDetectetAdress    := -1;
			utQuery.uiReadAddress   :=  0;
			utQuery.uiReadQuantity  :=  0;
		END_IF;
        xIsLinked               := FALSE;     
        xJobDone                := FALSE;
        xDataAvailable          := FALSE;
        xIsQuerryReady          := FALSE;
        xIsLocked               := FALSE; 
		utResponse.bUnitId		:= 0;   
		utResponse.bFunctionCode:= 0;       
        utResponse.uiAddress    := 0;
        utResponse.uiQuantity   := 0;
        metCheckToUnlinkUnlock  := TRUE;
        metAnalytic();
    END_IF;
END_IF;
END_METHOD

METHOD metCheckQuerryAdr : BOOL
VAR_INPUT
    wAdressIn        :   WORD;
    uiQuantityIn     :   UINT;
    pByte            :   POINTER TO BYTE;
    wOffset          :   WORD;                  // Pointer Offset wenn Tcp WORD Array > 123 or Byte Array > 1968  | Serial Word Array > 68 or Byte Arry > 123       
END_VAR
(* Check if Locked *)
IF NOT xIsLocked AND NOT xIsQuerryReady THEN
    (* Check if Linked *)
    IF NOT xIsLinked THEN  
        metMaxQuantity();
        IF uiQuantityIn <= wMaxQuantity AND diSandwichAdress = wAdressIn OR diSandwichAdress = -1 THEN  
            IF diFirstDetectetAdress = -1 THEN
                diFirstDetectetAdress := wAdressIn;
            END_IF;  
            xIsLinked           := TRUE;
            diSandwichAdress    := -1;
            wStartAdress        := wAdressIn;
            uiQuantity          := uiQuantityIn;
            wStopAdress         := wStartAdress + uiQuantity - 1; 
            metSetQuerry();  
            IF bFunctionCode = 6 OR bFunctionCode = 5 OR bFunctionCode = 16 OR bFunctionCode = 15 THEN
                metSetWriteWord(wAdressIn,uiQuantityIn,xIsBoolQuerry,pByte,wOffset);
            END_IF;
            metCheckQuerryAdr   := TRUE; 
        END_IF;
    ELSE
        (* Task überschnitt verhindern *)
        IF wAdressIn = diFirstDetectetAdress  THEN
            xIsQuerryReady := TRUE;
        ELSIF uiQuantity = wMaxQuantity THEN
            xIsQuerryReady := TRUE;
		ELSE
            (* Add if Adr is next to linked *)
            IF uiQuantity + uiQuantityIn <= wMaxQuantity AND wAdressIn = wStopAdress + 1 THEN
                uiQuantity          := uiQuantity + uiQuantityIn;  
                wStopAdress         := wStartAdress + uiQuantity - 1;  
                metSetQuerry();     
                IF bFunctionCode = 6 OR bFunctionCode = 5 OR bFunctionCode = 16 OR bFunctionCode = 15 THEN
                    metSetWriteWord(wAdressIn,uiQuantityIn,xIsBoolQuerry,pByte,wOffset);
                END_IF;
                metCheckQuerryAdr   := TRUE; 
            (* Check if Adr is in Range *)       
            ELSIF wAdressIn >= wStartAdress AND wAdressIn <= wStopAdress THEN
                metCheckQuerryAdr := TRUE;   
            (* Sandwich Adresse ausfindig machen Bsp: 23|24|25|16|26|27 = 16 Sandwich*)  
            ELSIF wAdressIn <= wStartAdress THEN
                diSandwichAdress := wAdressIn;
            END_IF;
        END_IF;
	END_IF;
ELSE
    (* Wait Till Data Available *)
    IF xJobDone THEN
        IF xDataAvailable THEN
            metGetResponse(wAdressIn,uiQuantityIn,xIsBoolQuerry,pByte,wOffset);
        END_IF;  
        metCheckToUnlinkUnlock(wAdressIn,uiQuantityIn);  
	END_IF;  
END_IF;
END_METHOD

METHOD metLock : BOOL
VAR_INPUT
END_VAR
xIsLocked := TRUE;
END_METHOD

PROPERTY proAllJobsDone : BOOL
SET
xAllJobsDone := proAllJobsDone;
END_SET
GET
proAllJobsDone := xAllJobsDone;
END_GET
END_PROPERTY

METHOD PRIVATE metSetQuerry : BOOL
VAR_INPUT
END_VAR
utQuery.bUnitId         := bUnitId;
utQuery.bFunctionCode   := bFunctionCode;
utQuery.uiReadAddress   := wStartAdress;
utQuery.uiReadQuantity  := uiQuantity;
utQuery.uiWriteAddress  := wStartAdress;
utQuery.uiWriteQuantity := uiQuantity;
END_METHOD

METHOD PRIVATE metSetWriteWord : BOOL
VAR_INPUT
    wAdressIn        :   WORD;
    uiQuantityIn     :   UINT;
    xIsBoolQuerry    :   BOOL;              // TRUE = Bool Querry    
    pByte            :   POINTER TO WORD;
    wOffset          :   WORD;               // Pointer Offset wenn WORD Array > 123 or Byte Array > 1968     
END_VAR
IF xIsBoolQuerry THEN 
    metQuerryAyBoolToAyWord(wAdressIn,uiQuantityIn,wOffset,pByte);
ELSE
    metQuerryAyWordToAyWord(wAdressIn,uiQuantityIn,wOffset,pByte);
END_IF
END_METHOD

METHOD PRIVATE metGetResponse : BOOL
VAR_INPUT
    wAdressIn        :   WORD;
    uiQuantityIn     :   UINT;
    xIsBoolQuerry    :   BOOL;                  // TRUE = Bool Querry
    pByte            :   POINTER TO BYTE;
    wOffset          :   WORD;                  // Pointer Offset wenn WORD Array > 123 or Byte Array > 1968             
END_VAR
IF eErrorCurrent = WagoAppPlcModbus.eErrorModbus.OK AND utResponse.uiQuantity > 0 THEN
    IF utResponse.bFunctionCode <> 5 AND utResponse.bFunctionCode <> 6 AND utResponse.bFunctionCode <> 15 AND utResponse.bFunctionCode <> 16 THEN
        IF wAdressIn >= utResponse.uiAddress AND wAdressIn + uiQuantityIn <= utResponse.uiAddress + utResponse.uiQuantity THEN    
            IF xIsBoolQuerry THEN 
                metResponsAyWordToAyBool(wAdressIn,uiQuantityIn,wOffset,pByte);
            ELSE
                metResponsAyWordToAyWord(wAdressIn,uiQuantityIn,wOffset,pByte);
            END_IF;
        END_IF;
    END_IF;
END_IF;
END_METHOD

METHOD PRIVATE metQuerryAyWordToAyWord : BOOL
VAR_INPUT
    wAdressIn   :   WORD;
    uiQuantity  :   UINT;
    wOffset     :   WORD;
    pWord       :   POINTER TO WORD;    
END_VAR
VAR
    uiFor       :   UINT;
    pTarget     :   POINTER TO WORD;
END_VAR
(* Copy Word to Word Pointer *)
IF pWord <> 0 THEN
    FOR uiFor := 0 TO uiQuantity - 1 DO 
        pTarget  := pWord + (uiFor + wOffset) * 2;  // 2 = 2Byte
        utQuery.awWriteData[wAdressIn - utQuery.uiWriteAddress + uiFor] := pTarget^;
    END_FOR;   
END_IF;
END_METHOD

METHOD PRIVATE metQuerryAyBoolToAyWord : BOOL
VAR_INPUT
    wAdressIn       :   WORD;
    uiQuantity      :   UINT;
    wOffset         :   WORD;
    pByte           :   POINTER TO BYTE;    
END_VAR
VAR
    uiFor           :   UINT;
    usiCountWords   :   USINT; 
    pTarget         :   POINTER TO BYTE;
    wTempValue      :   WORD;
    wOffsetQuerry   :   WORD;
    wOffsetBit      :   WORD;
END_VAR
(* Transfaire Array of Byte to Word Array Modbus format *)
FOR uiFor := 0 TO uiQuantity - 1 DO
    (* Offset of Bit *)
    wOffsetBit    := (wAdressIn - utQuery.uiWriteAddress) MOD 16;
    (* Offset of Word Array *)
    IF wOffsetBit > 0 THEN
        wOffsetQuerry := (((wAdressIn - utQuery.uiWriteAddress) - wOffsetBit) / 16 );    
    ELSE
        wOffsetQuerry := (wAdressIn - utQuery.uiWriteAddress) / 16;
	END_IF;
    (* Get Overlaping Value *)
    IF uiFor <= wOffsetBit AND wOffsetBit <> 0 THEN
        wTempValue := utQuery.awWriteData[wOffsetQuerry];
    END_IF;
    (* Set Values *)
    IF uiFor MOD 16 = 0 AND uiFor > 0 THEN
        usiCountWords := usiCountWords + 1;
        wOffsetBit    := 0; // Reset Offset after Word Switch
    END_IF
    pTarget  := pByte + (uiFor + wOffset) * 1;    // 1 = 1Byte Bool needs 1 Byte drive not 1 Bit
    IF TO_BOOL(pTarget^) THEN 
        wTempValue  := wTempValue + TO_WORD(EXPT(2,wOffsetBit + uiFor - (usiCountWords * 16)));
    END_IF;
    utQuery.awWriteData[LIMIT(LOWER_BOUND(utQuery.awWriteData,1), wOffsetQuerry + usiCountWords,UPPER_BOUND(utQuery.awWriteData,1))] := wTempValue;    
END_FOR;
END_METHOD

METHOD PRIVATE metResponsAyWordToAyBool : BOOL
VAR_INPUT
    wAdressIn       :   WORD;
    uiQuantity      :   UINT;
    wOffset         :   WORD;
    pByte           :   POINTER TO BYTE;    
END_VAR
VAR
    uiFor           :   UINT;
    usiCountWords   :   USINT; 
    pTarget         :   POINTER TO BYTE;
    wTempValue      :   WORD;
    wOffsetQuerry   :   WORD;
    wOffsetBit      :   WORD;
END_VAR
(* Transfaire Array of Byte to Word Array Modbus format *)
FOR uiFor := 0 TO uiQuantity - 1 DO
    (* Offset of Bit *)
    wOffsetBit    := (wAdressIn - utResponse.uiAddress) MOD 16;
    (* Offset of Word Array *)
    IF wOffsetBit > 0 THEN
        wOffsetQuerry := (((wAdressIn - utResponse.uiAddress) - wOffsetBit) / 16);    
    ELSE
        wOffsetQuerry := (wAdressIn - utResponse.uiAddress)/16;
	END_IF;
    (* Get Overlaping Value *)
    IF uiFor <= wOffsetBit AND wOffsetBit <> 0 THEN
        wTempValue := utResponse.awData[wOffsetQuerry];
    END_IF;
    (* Set Values *)
    IF uiFor MOD 16 = 0 AND uiFor > 0 THEN
        usiCountWords := usiCountWords + 1;
        wOffsetBit    := 0; // Reset Offset after Word Switch
    END_IF
    pTarget  := pByte + (uiFor + wOffset) * 1;    // 1 = 1Byte Bool needs 1 Byte drive not 1 Bit
    pTarget^ := fcWordBitToByte(utResponse.awData[LIMIT(LOWER_BOUND(utResponse.awData,1),wOffsetQuerry + usiCountWords,UPPER_BOUND(utResponse.awData,1))],TO_USINT(woffsetBit + (uiFor-(16*usiCountWords))));
END_FOR;
END_METHOD

METHOD PRIVATE metResponsAyWordToAyWord : BOOL
VAR_INPUT
    wAdressIn   :   WORD;
    uiQuantity  :   UINT;
    wOffset     :   WORD;
    pWord       :   POINTER TO WORD;    
END_VAR
VAR
    uiFor       :   UINT;
    pTarget     :   POINTER TO WORD;
END_VAR
(* Copy Word to Word Pointer *)
IF pWord <> 0 THEN
    FOR uiFor := 0 TO uiQuantity - 1 DO 
        pTarget  := pWord + (uiFor + wOffset) * 2;  // 2 = 2Byte
        pTarget^ := utResponse.awData[wAdressIn - utResponse.uiAddress + uiFor];
    END_FOR;   
END_IF;
END_METHOD

METHOD metCallAfterResponse : BOOL
VAR_INPUT
    xError  :   BOOL;
    uiID    :   UINT;
END_VAR
IF NOT xJobDone THEN
    (* On Error *)
    IF xError OR utResponse.wError <> 0 THEN
        (* Erster Error Registrieren *)
        IF diErrorAdress = -1 OR eError = 0 THEN
            diErrorAdress   := wStartAdress;
            IF xError THEN
                eError          := uiID;
                eErrorCurrent   := uiID;
            ELSE
                eError          := utResponse.wError;
                eErrorCurrent   := utResponse.wError;            
            END_IF;
        ELSE
            (* Aktuelle Error *)
            IF xError THEN
                eErrorCurrent   := uiID;
            ELSE
                eErrorCurrent   := utResponse.wError;            
            END_IF;    
        END_IF;      
    ELSE
        IF wStartAdress = diErrorAdress THEN
            eError          := utResponse.wError;
            diErrorAdress   := -1;
		END_IF
        eErrorCurrent  := utResponse.wError;
        xDataAvailable := TRUE;
    END_IF;	
    xJobDone     := TRUE;    
	fbTimeDiscareJob.Start();
END_IF;
END_METHOD

//FB_Init ist immer implizit verfügbar und wird primär für die Initialisierung verwendet.
//Der Rückgabewert wird nicht ausgewertet. Für gezielte Einflussnahme können Sie
//die Methoden explizit deklarieren und darin mit dem Standard-Initialisierungscode 
//zusätzlichen Code bereitstellen. Sie können den Rückgabewert auswerten.
METHOD FB_Init: BOOL
VAR_INPUT    
bInitRetains: BOOL; // TRUE: Die Retain-Variablen werden initialisiert (Reset warm / Reset kalt)    
bInCopyCode: BOOL;  // TRUE: Die Instanz wird danach in den Kopiercode kopiert (Online-Change)
END_VAR
VAR
    diFor : DINT;
END_VAR
xIsLinked               := FALSE;   
xIsLocked               := FALSE;   
xJobDone                := FALSE;   
xAllJobsDone            := FALSE;   
diSandwichAdress        := -1;
diErrorAdress           := -1;
eError                  :=  0;
eErrorCurrent           :=  0;
wCountJobs              :=  0;
wCountJobsTemp          :=  0;
diFirstDetectetAdress   := -1;
diLastDetectetAdress    := -1;
diTempDetectetAdress    := -1;
utQuery.uiReadAddress   :=  0;
utQuery.uiReadQuantity  :=  0;
END_METHOD

METHOD PRIVATE metAnalytic : BOOL
VAR_INPUT
END_VAR
IF xCheckLastAdr AND wStartAdress <> diFirstDetectetAdress THEN
	metResetMissingLastAdr();
	xCheckLastAdr := TRUE;
END_IF
IF wStartAdress = diFirstDetectetAdress THEN
    IF xFirstRequestDone THEN
        IF diLastDetectetAdress = -1 THEN
            IF diTempDetectetAdress = -1 THEN
                diLastDetectetAdress := diFirstDetectetAdress;
            ELSE
                diLastDetectetAdress := diTempDetectetAdress;
            END_IF
            ltMessung       := fbTIME.Stop();   
            wCountJobs      := wCountJobsTemp;
            wCountJobsTemp  := 0; 
            xAllJobsDone    := TRUE;
		ELSE
			IF NOT xCheckLastAdr THEN
				metResetMissingLastAdr();
			ELSE
				xCheckLastAdr := FALSE;
			END_IF;
			xCheckFirstAdr := TRUE;
        END_IF;
        fbTIME.Start();   
     ELSE
         xFirstRequestDone := TRUE;
		 xCheckFirstAdr := TRUE;
		 xCheckLastAdr	:= FALSE;
	 END_IF;
ELSE
    diTempDetectetAdress := wStartAdress;  
END_IF; 

wCountJobsTemp := wCountJobsTemp + 1;

IF wStartAdress = diLastDetectetAdress AND xFirstRequestDone THEN   
    ltMessung       := fbTIME.Stop();   
    wCountJobs      := wCountJobsTemp;
    wCountJobsTemp  := 0; 
    xAllJobsDone    := TRUE;
	IF NOT xCheckFirstAdr THEN
		metResetMissingFirstAdr();
	ELSE
		xCheckFirstAdr := FALSE;
	END_IF;
	xCheckLastAdr := TRUE;
END_IF;   

IF xFirstRequestDone AND ((xCheckLastAdr AND xCheckFirstAdr) OR (NOT xCheckLastAdr AND NOT xCheckFirstAdr)) THEN
	metResetMissingFirstAdr();
	metResetMissingLastAdr();
END_IF;
END_METHOD

METHOD metMaxQuantity : WORD;
IF xIsSerialJob THEN
    IF xIsBoolQuerry THEN
        IF bFunctionCode = 15 THEN
            wMaxQuantity := Parameter.wQuantityWriteSerialBool;
		ELSIF bFunctionCode = 5 THEN
			wMaxQuantity := 1;
        ELSE
            wMaxQuantity := Parameter.wQuantityReadSerialBool;
        END_IF;
    ELSE
        IF bFunctionCode = 16 THEN
            wMaxQuantity := Parameter.wQuantityWriteSerialWord;
		ELSIF bFunctionCode = 6 THEN
			wMaxQuantity := 1;
        ELSE
            wMaxQuantity := Parameter.wQuantityReadSerialWord;
        END_IF;        
	END_IF
ELSE
    IF xIsBoolQuerry THEN
        IF bFunctionCode = 15 THEN
            wMaxQuantity := Parameter.wQuantityWriteTcpBool;
		ELSIF bFunctionCode = 5 THEN
			wMaxQuantity := 1;		
        ELSE
            wMaxQuantity := Parameter.wQuantityReadTcpBool;
        END_IF;
    ELSE
        IF bFunctionCode = 16 THEN
            wMaxQuantity := Parameter.wQuantityWriteTcpWord;
		ELSIF bFunctionCode = 6 THEN
			wMaxQuantity := 1;
        ELSE
            wMaxQuantity := Parameter.wQuantityReadTcpWord;
        END_IF;        
	END_IF    
END_IF
END_METHOD

METHOD metResetMissingLastAdr : BOOL
VAR_INPUT
END_VAR
xFirstRequestDone 		:= FALSE;
diLastDetectetAdress    := -1;
diTempDetectetAdress    := wStartAdress;
wCountJobsTemp			:= 0;
END_METHOD

METHOD metResetMissingFirstAdr : BOOL
VAR_INPUT
END_VAR
diFirstDetectetAdress   := -1;
diTempDetectetAdress    := -1;
xFirstRequestDone 		:= FALSE;
wCountJobsTemp			:= 0;
END_METHOD

END_FUNCTION_BLOCK

// 30 Program Organization Units/CONVERTER/fcWordBitToByte
FUNCTION fcWordBitToByte : BYTE
VAR_INPUT
    wIn     :   WORD;
    usiBit  :   USINT;
END_VAR
VAR
    wTemp   :   WORD;
END_VAR

IF usiBit >= 0 AND usiBit <= 15 THEN
    wTemp := SHL(wIn,15-usiBit);
    wTemp := SHR(wTemp,15);
    fcWordBitToByte := TO_BYTE(wTemp);
END_IF;

END_FUNCTION

// 30 Program Organization Units/CLIENT/NETWORK Client/UDP/fbMbUdpClient
FUNCTION_BLOCK fbMbUdpClient EXTENDS CtaSysBase.fbBASE IMPLEMENTS ITF_MbClient                  
VAR_OUTPUT                      
    xError                      : BOOL;
END_VAR
VAR    
	ITF_BMK 					: CtaAppBmk.ITF_BMK;	
	xComAktive                  : BOOL;
    (* Udp Client *)
    byUnitId                    : BYTE;
    fbMbClientUdp               : WagoAppPLCModbus.FbMbMasterUdp;
    
    (* Main State *)
    uiCountErrors               : UINT;   
    usiState                    : USINT := 1;
    fbTIMEFcs                   : CtaAppTime.fbTimeMeasurement;
    ltMessungFcs                : LTIME; 
    
    (* Scan Rate *)
    TON_ScanRate                : TON;
    tonDelayRead				: Standard.TON;
	tonDelayWrite				: Standard.TON;
	xTrigDelayRead				: BOOL;
	xTrigDelayWrite				: BOOL; 
    (* User Querry *)
    xTrigStart                  : BOOL;
    xTrigStopp                  : BOOL;
    xTrig                       : BOOL;
    utQueryTrig                 : typMbQuery    := (bUnitId         := byUnitId,
                                                    uiReadAddress   := 0,
                                                    uiReadQuantity  := 0,
                                                    bFunctionCode   := 1);    
    utResponseTrig              : typMbResponse; 
    ltMessungTrig               : LTIME;
    fbTIMETrig                  : CtaAppTime.fbTimeMeasurement;
    
    (* FC1 *)
    fbJobFc1                    : fbJOB;
    xTrigFc1                    : BOOL;
    fbTIMEFc1                   : CtaAppTime.fbTimeMeasurement;
    ltMessungFc1                : LTIME;      
    (* FC2 *)
    fbJobFc2                    : fbJOB;
    xTrigFc2                    : BOOL; 
    fbTIMEFc2                   : CtaAppTime.fbTimeMeasurement;
    ltMessungFc2                : LTIME;      
    (* FC3 *)
    fbJobFc3                    : fbJOB;
    xTrigFc3                    : BOOL;      
    fbTIMEFc3                   : CtaAppTime.fbTimeMeasurement;
    ltMessungFc3                : LTIME;          
    (* FC4 *)
    fbJobFc4                    : fbJOB;
    xTrigFc4                    : BOOL;      
    fbTIMEFc4                   : CtaAppTime.fbTimeMeasurement;
    ltMessungFc4                : LTIME;      
    (* FC5 *)
    fbJobFc5                    : fbJOB;
    xTrigFc5                    : BOOL;      
    fbTIMEFc5                   : CtaAppTime.fbTimeMeasurement;
    ltMessungFc5                : LTIME;      
    (* FC6 *)
    fbJobFc6                    : fbJOB;
    xTrigFc6                    : BOOL;      
    fbTIMEFc6                   : CtaAppTime.fbTimeMeasurement;
    ltMessungFc6                : LTIME;    
    (* FC15 *)
    fbJobFc15                   : fbJOB;
    xTrigFc15                   : BOOL;   
    fbTIMEFc15                  : CtaAppTime.fbTimeMeasurement;
    ltMessungFc15               : LTIME;     
    (* FC16 *)   
    fbJobFc16                   : fbJOB;             
    xTrigFc16                   : BOOL;
    fbTIMEFc16                  : CtaAppTime.fbTimeMeasurement;
    ltMessungFc16               : LTIME;      
(* FC43 *)   
    fbIdentifyObject			: WagoAppPlcModbus.FbIdentifyBaseObject;
	fbIdentifyMember3			: WagoAppPlcModbus.FbIdentifyMember_STRING(fbIdentifyObject,3);
	fbIdentifyMember4			: WagoAppPlcModbus.FbIdentifyMember_STRING(fbIdentifyObject,4);
	utIdentifyQuerry			: WagoAppPlcModbus.typMbQuery;
	utIdentifyResponse			: WagoAppPlcModbus.typMbResponse;           
    xTrigFc43                   : BOOL;
	xActiveFc43					: BOOL;
	xDoneFc43					: BOOL;
	tTimeOutFc43				: TIME;
    fbTIMEFc43                  : CtaAppTime.fbTimeMeasurement;
    ltMessungFc43               : LTIME; 
    (* Parameter *)
    fbConfigFile                : CtaSysConfig.fbConfigFile;
    scParameter                 : scUdpClientParameter;
END_VAR

(* Config *)
actConfig();
(* Unit ID *)
byUnitId := scParameter.fbbyUnitId.byValue;
IF scParameter.fbxEnable.xValue AND byUnitId <> 0 THEN
	(* Delay *)
	actDelay();
	(* FC1 *)
	actFC01();
	(* FC2 *)
	actFC02();
	(* FC3 *)
	actFC03();
	(* FC4 *)
	actFC04();
	(* FC5 *)
	actFC05();
	(* FC6 *)
	actFC06();	
	(* FC15 *)
	actFC15();
	(* FC16 *)
	actFC16(); 
	(* User Querry *)
	actFcUserQuerry();
END_IF;
	IF usiState >= 8 OR usiState = 0 THEN
		(* Check if all Jobs Done *)
        IF  fbJobFc1.xAllJobsDone  AND
            fbJobFc2.xAllJobsDone  AND
            fbJobFc3.xAllJobsDone  AND
            fbJobFc4.xAllJobsDone  AND
            fbJobFc5.xAllJobsDone  AND
            fbJobFc6.xAllJobsDone  AND			
            fbJobFc15.xAllJobsDone AND
            fbJobFc16.xAllJobsDone THEN
			(*Scan Rate *)
			TON_ScanRate(IN := NOT TON_ScanRate.Q,
						 PT := scParameter.fbtScanRate.tValue);
						 
			IF TON_ScanRate.Q THEN
                fbJobFc1.proAllJobsDone  := FALSE;
                fbJobFc2.proAllJobsDone  := FALSE;   
                fbJobFc3.proAllJobsDone  := FALSE;  
                fbJobFc4.proAllJobsDone  := FALSE;   
                fbJobFc5.proAllJobsDone  := FALSE;  
                fbJobFc6.proAllJobsDone  := FALSE; 	
                fbJobFc15.proAllJobsDone := FALSE;  
                fbJobFc16.proAllJobsDone := FALSE; 
				usiState := 1;
				(* Timer stopp *) 
				ltMessungFcs := fbTIMEFcs.stop();             
				(* Timer start *) 
				fbTIMEFcs.Start();      
			END_IF;        
		ELSE    
			usiState := 1;
		END_IF;   
	END_IF;
	xComAktive := fbJobFc1.wCountJobs  <> 0 OR 
				  fbJobFc2.wCountJobs  <> 0 OR
				  fbJobFc3.wCountJobs  <> 0 OR 
				  fbJobFc4.wCountJobs  <> 0 OR 
				  fbJobFc15.wCountJobs <> 0 OR
				  fbJobFc16.wCountJobs <> 0 ;  
	(* Get Errors *)
	xError :=  fbJobFc1.eError <> WagoAppPlcModbus.eErrorModbus.OK OR 
			   fbJobFc2.eError <> WagoAppPlcModbus.eErrorModbus.OK OR 
			   fbJobFc3.eError <> WagoAppPlcModbus.eErrorModbus.OK OR 
			   fbJobFc4.eError <> WagoAppPlcModbus.eErrorModbus.OK OR 
			   fbJobFc5.eError <> WagoAppPlcModbus.eErrorModbus.OK OR
			   fbJobFc6.eError <> WagoAppPlcModbus.eErrorModbus.OK OR
			  fbJobFc15.eError <> WagoAppPlcModbus.eErrorModbus.OK OR 
			  fbJobFc16.eError <> WagoAppPlcModbus.eErrorModbus.OK OR
			  fbConfigFile.xError;
			  
	IF NOT xError THEN
	   uiCountErrors := 0;
	END_IF;

ACTION actFC16:
(* Trig FC16 *)
IF fbJobFc16.xIsLinked AND fbJobFc16.xIsQuerryReady AND NOT fbJobFc16.xIsLocked AND NOT fbJobFc16.xAllJobsDone AND tonDelayWrite.Q THEN
    fbJobFc16.metLock();
    xTrigFc16       := TRUE;
    fbTIMEFc16.Start();
ELSIF usiState = 8 AND (NOT fbJobFc16.xIsLinked OR fbJobFc16.xAllJobsDone) THEN
    usiState                    := usiState + 1; 
    fbJobFc16.proAllJobsDone    := TRUE;   
END_IF
(* Send Querry *)
IF usiState = 8  AND xTrigFc16 THEN
	xTrigDelayWrite := FALSE;
    fbMbClientUdp              (xConnect    := TRUE,
                                sHost       := scParameter.fbstIp.stValue,
                                wPort       := scParameter.fbwPort.wValue,
                                eFrameType  := WagoAppPlcModbus.eMbFrameType.ETHERNET,
                                tTimeOut    := scParameter.fbtTimeOut.tValue,
                                utQuery     := fbJobFc16.utQuery,
                                xTrigger    := xTrigFc16,
                                utResponse  := fbJobFc16.utResponse);       
END_IF;
(* Get Response *) 
IF usiState = 8 AND NOT xTrigFc16 AND fbJobFc16.xIsLocked AND NOT fbJobFc16.xJobDone THEN
    usiState            := usiState + 1;
    ltMessungFc16       := fbTIMEFc16.Stop();
    metCheckOnError();
    fbJobFc16.metCallAfterResponse(fbMbClientUdp.xError,fbMbClientUdp.oStatus.uiID);
END_IF;
END_ACTION

METHOD PRIVATE FINAL metCheckOnError : BOOL
VAR_INPUT
END_VAR
IF fbMbClientUdp.xError THEN
    uiCountErrors  := uiCountErrors + 1;
    metCheckOnError := TRUE;
END_IF
END_METHOD

ACTION actFcUserQuerry:
IF xTrigStart AND usiState = 7 THEN
    xTrig       := TRUE;
    xTrigStart  := FALSE;
    xTrigStopp  := TRUE;
    fbTIMETrig.Start();
    utQueryTrig.bUnitId := scParameter.fbbyUnitId.byValue;
ELSIF NOT xTrig AND usiState = 7 THEN
    usiState := usiState + 1;        
END_IF;
IF usiState = 7 THEN
    fbMbClientUdp              (xConnect    := TRUE,
                                sHost       := scParameter.fbstIp.stValue,
                                wPort       := scParameter.fbwPort.wValue,
                                eFrameType  := WagoAppPlcModbus.eMbFrameType.ETHERNET,
                                tTimeOut    := scParameter.fbtTimeOut.tValue,
                                utQuery     := utQueryTrig,
                                xTrigger    := xTrig,
                                utResponse  := utResponseTrig);     
END_IF;  
                              
IF NOT xTrig AND xTrigStopp THEN
    ltMessungTrig := fbTIMETrig.Stop();
    xTrigStopp := FALSE;
    usiState := usiState + 1;
END_IF;
END_ACTION

METHOD FINAL metFc4ReadInputRegister
VAR_INPUT
    wADR                :   WORD;
    pWord               :   POINTER TO WORD;
    uiQuantity          :   UINT;               // Anzahl Words Max 123
    wOffset             :   WORD;               // Pointer Offset wenn WORD Array > 123   
END_VAR
VAR
    diCurrentJop        :   DINT;
    uiFor               :   UINT;
    pBaseAdr            :   POINTER TO WORD;
END_VAR
(* Limit Read Input Register *)
uiQuantity := LIMIT(1,uiQuantity,123);
(* Check if valid Pointer and Adress *)
IF pWord <> 0 AND wOffset + uiQuantity <= 16#FFFF + 1 AND wADR <= 16#FFFF THEN
    (* Link Adress *)
    fbJobFc4.bUnitId       := byUnitId;   
    fbJobFc4.bFunctionCode := 4;
    fbJobFc4.xIsBoolQuerry := FALSE;
    fbJobFc4.xIsSerialJob  := FALSE;     
    fbJobFc4.metCheckQuerryAdr(wADR,uiQuantity,pWord,wOffset);        
END_IF;
END_METHOD

ACTION actFC04:
(* Trig FC4 *)
IF fbJobFc4.xIsLinked AND fbJobFc4.xIsQuerryReady AND NOT fbJobFc4.xIsLocked AND NOT fbJobFc4.xAllJobsDone AND tonDelayRead.Q THEN
    fbJobFc4.metLock();
    xTrigFc4       := TRUE;
    fbTIMEFc4.Start();
ELSIF usiState = 4 AND (NOT fbJobFc4.xIsLinked OR fbJobFc4.xAllJobsDone) THEN
    usiState                := usiState + 1;    
    fbJobFc4.proAllJobsDone := TRUE;
END_IF
(* Send Querry *)
IF usiState = 4 AND xTrigFc4 THEN
	xTrigDelayRead 	:= FALSE;
    fbMbClientUdp              (xConnect    := TRUE,
                                sHost       := scParameter.fbstIp.stValue,
                                wPort       := scParameter.fbwPort.wValue,
                                eFrameType  := WagoAppPlcModbus.eMbFrameType.ETHERNET,
                                tTimeOut    := scParameter.fbtTimeOut.tValue,
                                utQuery     := fbJobFc4.utQuery,
                                xTrigger    := xTrigFc4,
                                utResponse  := fbJobFc4.utResponse);       
END_IF;
(* Get Response *) 
IF usiState = 4 AND NOT xTrigFc4 AND fbJobFc4.xIsLocked AND NOT fbJobFc4.xJobDone THEN 
    usiState            := usiState + 1;
    ltMessungFc4        := fbTIMEFc4.Stop();
    metCheckOnError();
    fbJobFc4.metCallAfterResponse(fbMbClientUdp.xError,fbMbClientUdp.oStatus.uiID);
END_IF;
END_ACTION

ACTION actFC02:
(* Trig FC2 *)
IF fbJobFc2.xIsLinked AND fbJobFc2.xIsQuerryReady AND NOT fbJobFc2.xIsLocked AND NOT fbJobFc2.xAllJobsDone AND tonDelayRead.Q THEN
    fbJobFc2.metLock();
    xTrigFc2       := TRUE;
    fbTIMEFc2.Start();
ELSIF usiState = 2 AND (NOT fbJobFc2.xIsLinked OR fbJobFc2.xAllJobsDone) THEN
    usiState                := usiState + 1;    
    fbJobFc2.proAllJobsDone := TRUE;
END_IF
(* Send Querry *)
IF usiState = 2 AND xTrigFc2 THEN
	xTrigDelayRead 	:= FALSE;
    fbMbClientUdp              (xConnect    := TRUE,
                                sHost       := scParameter.fbstIp.stValue,
                                wPort       := scParameter.fbwPort.wValue,
                                eFrameType  := WagoAppPlcModbus.eMbFrameType.ETHERNET,
                                tTimeOut    := scParameter.fbtTimeOut.tValue,
                                utQuery     := fbJobFc2.utQuery,
                                xTrigger    := xTrigFc2,
                                utResponse  := fbJobFc2.utResponse);       
END_IF;
(* Get Response *) 
IF usiState = 2 AND NOT xTrigFc2 AND fbJobFc2.xIsLocked AND NOT fbJobFc2.xJobDone THEN  
    usiState            := usiState + 1;
    ltMessungFc2        := fbTIMEFc2.Stop();
    metCheckOnError();
    fbJobFc2.metCallAfterResponse(fbMbClientUdp.xError,fbMbClientUdp.oStatus.uiID);
END_IF;
END_ACTION

METHOD FINAL metFc2ReadDiscretInput
VAR_INPUT
    wADR                :   WORD;
    pByte               :   POINTER TO BYTE;
    uiQuantity          :   UINT;               // Anzahl BOOL Max 1968
    wOffset             :   WORD;               // Pointer Offset wenn BOOL Array > 1968    
END_VAR
VAR
    diCurrentJop        :   DINT;
    uiFor               :   UINT;
    usiCountWords       :   UINT;    
    wTempValue          :   WORD;
    pBaseAdr            :   POINTER TO BYTE;
END_VAR
(* Limit Discret Inputs *)
uiQuantity := LIMIT(1,uiQuantity,1968);
(* Check if valid Pointer and Adress *)
IF pByte <> 0 AND wOffset + uiQuantity <= 16#FFFF + 1 AND wADR <= 16#FFFF THEN
    (* Link Adress *)
    fbJobFc2.bUnitId       := byUnitId;
    fbJobFc2.bFunctionCode := 2;
    fbJobFc2.xIsBoolQuerry := TRUE;
    fbJobFc2.xIsSerialJob  := FALSE;    
    fbJobFc2.metCheckQuerryAdr(wADR,uiQuantity,pByte,wOffset);    
END_IF;
END_METHOD

//FB_Init ist immer implizit verfügbar und wird primär für die Initialisierung verwendet.
//Der Rückgabewert wird nicht ausgewertet. Für gezielte Einflussnahme können Sie
//die Methoden explizit deklarieren und darin mit dem Standard-Initialisierungscode 
//zusätzlichen Code bereitstellen. Sie können den Rückgabewert auswerten.
METHOD FB_Init: BOOL
VAR_INPUT    
bInitRetains: BOOL; // TRUE: Die Retain-Variablen werden initialisiert (Reset warm / Reset kalt)    
bInCopyCode: BOOL;  // TRUE: Die Instanz wird danach in den Kopiercode kopiert (Online-Change)
END_VAR
xTrigFc1    := FALSE;
xTrigFc2    := FALSE;
xTrigFc3    := FALSE;
xTrigFc4    := FALSE;
xTrigFc15   := FALSE;
xTrigFc16   := FALSE;
xTrig       := FALSE;
usiState    := 0;
END_METHOD

METHOD FINAL metFc1ReadCoils
VAR_INPUT
    wADR                :   WORD;
    pByte               :   POINTER TO BYTE;
    uiQuantity          :   UINT;               // Anzahl Coils Max 1968
    wOffset             :   WORD;               // Pointer Offset wenn BOOL Array > 1968     
END_VAR
VAR
    diCurrentJop        :   DINT;
    uiFor               :   UINT;
    usiCountWords       :   UINT;
    wTempValue          :   WORD;
END_VAR
(* Limit Coils *)
uiQuantity := LIMIT(1,uiQuantity,1968);
(* Check if valid Pointer and Adress *)
IF pByte <> 0 AND wOffset + uiQuantity <= 16#FFFF + 1 AND wADR <= 16#FFFF THEN
    (* Link Adress *)
    fbJobFc1.bUnitId       := byUnitId;
    fbJobFc1.bFunctionCode := 1;
    fbJobFc1.xIsBoolQuerry := TRUE;
    fbJobFc1.xIsSerialJob  := FALSE;    
    fbJobFc1.metCheckQuerryAdr(wADR,uiQuantity,pByte,wOffset);        
END_IF;
END_METHOD

METHOD FINAL metFc15WriteMultipleCoil
VAR_INPUT
    wADR                :   WORD;
    pByte               :   POINTER TO BYTE;
    uiQuantity          :   UINT;               // Anzahl Coils Max 1968   
    wOffset             :   WORD;               // Pointer Offset wenn BOOL Array > 1968     
END_VAR
VAR
    diCurrentJop        :   DINT;
    uiFor               :   UINT;
    usiCountWords       :   UINT;
    wTempValue          :   WORD;    
END_VAR
(* Limit Write Multiple Coil *)
uiQuantity := LIMIT(1,uiQuantity,1968);
(* Check if valid Pointer and Adress *)
IF pByte <> 0 AND wOffset + uiQuantity <= 16#FFFF + 1 AND wADR <= 16#FFFF THEN
    (* Link Adress *)
    fbJobFc15.bUnitId       := byUnitId;
    fbJobFc15.bFunctionCode := 15;
    fbJobFc15.xIsBoolQuerry := TRUE;
    fbJobFc15.xIsSerialJob  := FALSE;        
    fbJobFc15.metCheckQuerryAdr(wADR,uiQuantity,pByte,wOffset);    
END_IF;
END_METHOD

METHOD FINAL metFc16WriteHoldingRegisters
VAR_INPUT
    wADR                :   WORD;
    pWord               :   POINTER TO WORD;
    uiQuantity          :   UINT;               // Anzahl Words Max 123
    wOffset             :   WORD;               // Pointer Offset wenn Array > 123 WORD    
END_VAR
VAR
    diCurrentJop        :   DINT;
    uiFor               :   UINT;
END_VAR
(* Limit Write Holding Registers *)
uiQuantity := LIMIT(1,uiQuantity,123);
(* Check if valid Pointer and Adress *)
IF pWord <> 0 AND wOffset + uiQuantity <= 16#FFFF + 1 AND wADR <= 16#FFFF THEN
    (* Link Adress *)
    fbJobFc16.bUnitId       := byUnitId;
    fbJobFc16.bFunctionCode := 16;
    fbJobFc16.xIsBoolQuerry := FALSE;
    fbJobFc16.xIsSerialJob  := FALSE;    
    fbJobFc16.metCheckQuerryAdr(wADR,uiQuantity,pWord,wOffset);
END_IF;
END_METHOD

ACTION actFC01:
(* Trig FC1 *)
IF fbJobFc1.xIsLinked AND fbJobFc1.xIsQuerryReady AND NOT fbJobFc1.xIsLocked AND NOT fbJobFc1.xAllJobsDone AND tonDelayRead.Q THEN
    fbJobFc1.metLock();
    xTrigFc1       := TRUE;
    fbTIMEFc1.Start();
ELSIF usiState = 1 AND (NOT fbJobFc1.xIsLinked OR fbJobFc1.xAllJobsDone) THEN
    usiState                := usiState + 1;    
    fbJobFc1.proAllJobsDone := TRUE;
END_IF
(* Send Querry *)
IF usiState = 1 AND xTrigFc1 THEN
	xTrigDelayRead 	:= FALSE;
    fbMbClientUdp              (xConnect    := TRUE,
                                sHost       := scParameter.fbstIp.stValue,
                                wPort       := scParameter.fbwPort.wValue,
                                eFrameType  := WagoAppPlcModbus.eMbFrameType.ETHERNET,
                                tTimeOut    := scParameter.fbtTimeOut.tValue,
                                utQuery     := fbJobFc1.utQuery,
                                xTrigger    := xTrigFc1,
                                utResponse  := fbJobFc1.utResponse);       
END_IF;
(* Get Response *) 
IF usiState = 1 AND NOT xTrigFc1 AND fbJobFc1.xIsLocked AND NOT fbJobFc1.xJobDone THEN
    usiState            := usiState + 1;
    ltMessungFc1        := fbTIMEFc1.Stop();
    metCheckOnError();
    fbJobFc1.metCallAfterResponse(fbMbClientUdp.xError,fbMbClientUdp.oStatus.uiID);
END_IF;
END_ACTION

ACTION actFC03:
(* Trig FC3 *)
IF fbJobFc3.xIsLinked AND fbJobFc3.xIsQuerryReady AND NOT fbJobFc3.xIsLocked AND NOT fbJobFc3.xAllJobsDone AND tonDelayRead.Q THEN
    fbJobFc3.metLock();
    xTrigFc3       := TRUE;
    fbTIMEFc3.Start();
ELSIF usiState = 3 AND (NOT fbJobFc3.xIsLinked OR fbJobFc3.xAllJobsDone) THEN
    usiState                := usiState + 1;    
    fbJobFc3.proAllJobsDone := TRUE;
END_IF
(* Send Querry *)
IF usiState = 3 AND xTrigFc3 THEN
	xTrigDelayRead 	:= FALSE;
    fbMbClientUdp              (xConnect    := TRUE,
                                sHost       := scParameter.fbstIp.stValue,
                                wPort       := scParameter.fbwPort.wValue,
                                eFrameType  := WagoAppPlcModbus.eMbFrameType.ETHERNET,
                                tTimeOut    := scParameter.fbtTimeOut.tValue,
                                utQuery     := fbJobFc3.utQuery,
                                xTrigger    := xTrigFc3,
                                utResponse  := fbJobFc3.utResponse);       
END_IF;
(* Get Response *) 
IF usiState = 3 AND NOT xTrigFc3 AND fbJobFc3.xIsLocked AND NOT fbJobFc3.xJobDone THEN  
    usiState            := usiState + 1;
    ltMessungFc3        := fbTIMEFc3.Stop();
    metCheckOnError();
    fbJobFc3.metCallAfterResponse(fbMbClientUdp.xError,fbMbClientUdp.oStatus.uiID);
END_IF;
END_ACTION

ACTION actFC15:
(* Trig FC15 *)
IF fbJobFc15.xIsLinked AND fbJobFc15.xIsQuerryReady AND NOT fbJobFc15.xIsLocked AND NOT fbJobFc15.xAllJobsDone AND tonDelayWrite.Q THEN
    fbJobFc15.metLock();
    xTrigFc15       := TRUE;
    fbTIMEFc15.Start();
ELSIF usiState = 7 AND (NOT fbJobFc15.xIsLinked OR fbJobFc15.xAllJobsDone) THEN
    usiState                    := usiState + 1;  
    fbJobFc15.proAllJobsDone    := TRUE;  
END_IF
(* Send Querry *)
IF usiState = 7 AND xTrigFc15 THEN
	xTrigDelayWrite := FALSE;
    fbMbClientUdp              (xConnect    := TRUE,
                                sHost       := scParameter.fbstIp.stValue,
                                wPort       := scParameter.fbwPort.wValue,
                                eFrameType  := WagoAppPlcModbus.eMbFrameType.ETHERNET,
                                tTimeOut    := scParameter.fbtTimeOut.tValue,
                                utQuery     := fbJobFc15.utQuery,
                                xTrigger    := xTrigFc15,
                                utResponse  := fbJobFc15.utResponse);       
END_IF;
(* Get Response *) 
IF usiState = 7 AND NOT xTrigFc15 AND fbJobFc15.xIsLocked AND NOT fbJobFc15.xJobDone THEN      
    usiState            := usiState + 1;
    ltMessungFc15       := fbTIMEFc15.Stop();
    metCheckOnError();
    fbJobFc15.metCallAfterResponse(fbMbClientUdp.xError,fbMbClientUdp.oStatus.uiID);
END_IF;
END_ACTION

METHOD FINAL metFc3ReadHoldingRegister
VAR_INPUT
    wADR                :   WORD;
    pWord               :   POINTER TO WORD;
    uiQuantity          :   UINT;               // Anzahl Words Max 123
    wOffset             :   WORD;               // Pointer Offset wenn WORD Array > 123    
END_VAR
VAR
    diCurrentJop        :   DINT;
    uiFor               :   UINT;
    pBaseAdr            :   POINTER TO WORD;
END_VAR
(* Limit Holding Register *)
uiQuantity := LIMIT(1,uiQuantity,123);
(* Check if valid Pointer and Adress *)
IF pWord <> 0 AND wOffset + uiQuantity <= 16#FFFF + 1 AND wADR <= 16#FFFF THEN
    (* Link Adress *)
    fbJobFc3.bUnitId       := byUnitId;
    fbJobFc3.bFunctionCode := 3;
    fbJobFc3.xIsBoolQuerry := FALSE;
    fbJobFc3.xIsSerialJob  := FALSE;       
    fbJobFc3.metCheckQuerryAdr(wADR,uiQuantity,pWord,wOffset);     
END_IF;
END_METHOD

ACTION actConfig:
(* Config File *)
fbConfigFile();

scparameter.fbbyUnitId          (_usiParaNr :=  1, itfConfigFb := fbconfigFile , _MinInit := 0      ,_MaxInit := 247	 );
scparameter.fbstIp              (_usiParaNr :=  2, itfConfigFb := fbconfigFile );
scparameter.fbwPort             (_usiParaNr :=  3, itfConfigFb := fbconfigFile );
scparameter.fbtTimeOut          (_usiParaNr :=  4, itfConfigFb := fbconfigFile , _MinInit := T#500MS,_MaxInit := T#10M	 );
scparameter.fbtScanRate         (_usiParaNr :=  5, itfConfigFb := fbconfigFile , _MinInit := T#00MS ,_MaxInit := T#10M	 );
scParameter.fbtDelayRead		(_usiParaNr :=  6, itfConfigFb := fbconfigFile , _MinInit := T#1MS  ,_MaxInit := T#10M   );	
scParameter.fbtDelayWrite		(_usiParaNr :=  7, itfConfigFb := fbconfigFile , _MinInit := T#1MS  ,_MaxInit := T#10M   );
END_ACTION

ACTION actFC43:
(* Trig FC43 *)
IF usiState = 9 AND NOT xDoneFc43 AND NOT xActiveFc43 THEN
	xTrigFc43       	:= TRUE;
	xActiveFc43			:= TRUE;
	tTimeOutFc43		:= T#1S;
	utIdentifyQuerry.bUnitId			:= byUnitId;
	utIdentifyQuerry.bFunctionCode		:= 43;	
	utIdentifyQuerry.IIdentifyObject	:= fbIdentifyObject;	
    fbTIMEFc43.Start();
ELSIF usiState = 9 AND NOT xActiveFc43 THEN
    usiState                := usiState + 1; 
END_IF
(* Send Querry *)
IF usiState = 9 AND xTrigFc43 THEN
    fbMbClientUdp              (xConnect    := TRUE,
                                sHost       := scParameter.fbstIp.stValue,
                                wPort       := scParameter.fbwPort.wValue,
                                eFrameType  := WagoAppPlcModbus.eMbFrameType.ETHERNET,
                                tTimeOut    := tTimeOutFc43,
                                utQuery     := utIdentifyQuerry,
                                xTrigger    := xTrigFc43,
                                utResponse  := utIdentifyResponse);   
    	      
END_IF;
(* Get Response *) 
IF usiState = 9 AND NOT xTrigFc43 AND xActiveFc43 AND NOT xDoneFc43 THEN
    usiState            := usiState + 1;
    ltMessungFc43       := fbTIMEFc43.Stop();
	xActiveFc43 		:= FALSE;
	IF fbMbClientUdp.oStatus.uiID = 16#99 THEN
		xDoneFc43			:= FALSE;
	ELSE
		xDoneFc43			:= TRUE;
	END_IF;
END_IF;
END_ACTION

{attribute 'monitoring' := 'call'}
PROPERTY sProductCode : STRING(WagoAppPlcModbus.Parameter.MAX_IDENTIFICATION_MEMBER_LENGTH)
GET
sProductCode := fbIdentifyObject.sProductCode;
END_GET
END_PROPERTY

{attribute 'monitoring' := 'call'}
PROPERTY sVendorName : STRING(WagoAppPlcModbus.Parameter.MAX_IDENTIFICATION_MEMBER_LENGTH)
GET
sVendorName := fbIdentifyObject.sVendorName;
END_GET
END_PROPERTY

{attribute 'monitoring' := 'call'}
PROPERTY sMajorMinorRevision : STRING(WagoAppPlcModbus.Parameter.MAX_IDENTIFICATION_MEMBER_LENGTH)
GET
sMajorMinorRevision := fbIdentifyObject.sMajorMinorRevision;
END_GET
END_PROPERTY

PROPERTY proModBusOK : BOOL
GET
proModBusOK := xComAktive AND NOT xError;
END_GET
END_PROPERTY

METHOD FINAL metFc5WriteCoil
VAR_INPUT
    wADR                :   WORD;
    pByte               :   POINTER TO BYTE;
    uiQuantity          :   UINT;               // Anzahl Coils Max 2000   
    wOffset             :   WORD;               // Pointer Offset wenn BOOL Array > 125     
END_VAR
VAR
    diCurrentJop        :   DINT;
    uiFor               :   UINT;
    usiCountWords       :   UINT;
    wTempValue          :   WORD;    
END_VAR
(* Limit Write Multiple Coil *)
uiQuantity := LIMIT(1,uiQuantity,1);
(* Check if valid Pointer and Adress *)
IF pByte <> 0 AND wOffset + uiQuantity <= 16#FFFF + 1 AND wADR <= 16#FFFF THEN
    (* Link Adress *)
    fbJobFc5.bUnitId       := byUnitId;
    fbJobFc5.bFunctionCode := 5;
    fbJobFc5.xIsBoolQuerry := TRUE;
    fbJobFc5.xIsSerialJob  := TRUE;           
    fbJobFc5.metCheckQuerryAdr(wADR,uiQuantity,pByte,wOffset);    
END_IF;
END_METHOD

METHOD FINAL metFc6WriteHoldingRegister
VAR_INPUT
    wADR                :   WORD;
    pWord               :   POINTER TO WORD;
    uiQuantity          :   UINT;               // Anzahl Words Max 125
    wOffset             :   WORD;               // Pointer Offset wenn Array > 125 WORD    
END_VAR
VAR
    diCurrentJop        :   DINT;
    uiFor               :   UINT;
END_VAR
(* Limit Write Holding Registers *)
uiQuantity := LIMIT(1,uiQuantity,1);
(* Check if valid Pointer and Adress *)
IF pWord <> 0 AND wOffset + uiQuantity <= 16#FFFF + 1 AND wADR <= 16#FFFF THEN
    (* Link Adress *)
    fbJobFc6.bUnitId       := byUnitId;
    fbJobFc6.bFunctionCode := 6;
    fbJobFc6.xIsBoolQuerry := FALSE;
    fbJobFc6.xIsSerialJob  := FALSE;        
    fbJobFc6.metCheckQuerryAdr(wADR,uiQuantity,pWord,wOffset);
END_IF;
END_METHOD

ACTION actFC05:
(* Trig FC15 *)
IF fbJobFc5.xIsLinked AND fbJobFc5.xIsQuerryReady AND NOT fbJobFc5.xIsLocked AND NOT fbJobFc5.xAllJobsDone AND tonDelayWrite.Q THEN
    fbJobFc5.metLock();
    xTrigFc5       := TRUE;
    fbTIMEFc5.Start();
ELSIF usiState = 5 AND (NOT fbJobFc5.xIsLinked OR fbJobFc5.xAllJobsDone) THEN
    usiState                    := usiState + 1; 
    fbJobFc5.proAllJobsDone    := TRUE;   
END_IF
(* Send Querry *)
IF usiState = 5 AND xTrigFc5 THEN
	xTrigDelayWrite := FALSE;
    fbMbClientUdp              (xConnect    := TRUE,
                                sHost       := scParameter.fbstIp.stValue,
                                wPort       := scParameter.fbwPort.wValue,
                                eFrameType  := WagoAppPlcModbus.eMbFrameType.ETHERNET,
                                tTimeOut    := scParameter.fbtTimeOut.tValue,
                                utQuery     := fbJobFc5.utQuery,
                                xTrigger    := xTrigFc5,
                                utResponse  := fbJobFc5.utResponse);    
END_IF;
(* Get Response *) 
IF usiState = 5 AND NOT xTrigFc5 AND fbJobFc5.xIsLocked AND NOT fbJobFc5.xJobDone  THEN 
    usiState            := usiState + 1;
    ltMessungFc5       := fbTIMEFc5.Stop();
    metCheckOnError();
    fbJobFc6.metCallAfterResponse(fbMbClientUdp.xError,fbMbClientUdp.oStatus.uiID);
END_IF;
END_ACTION

ACTION actFC06:
(* Trig FC6 *)
IF fbJobFc6.xIsLinked AND fbJobFc6.xIsQuerryReady AND NOT fbJobFc6.xIsLocked AND NOT fbJobFc6.xAllJobsDone AND tonDelayWrite.Q THEN
    fbJobFc6.metLock();
    xTrigFc6       := TRUE;
    fbTIMEFc6.Start();
ELSIF usiState = 6 AND (NOT fbJobFc6.xIsLinked OR fbJobFc6.xAllJobsDone) THEN
    usiState                    := usiState + 1; 
    fbJobFc6.proAllJobsDone    := TRUE;   
END_IF
(* Send Querry *)
IF usiState = 6 AND xTrigFc6 THEN
	xTrigDelayWrite := FALSE;
    fbMbClientUdp              (xConnect    := TRUE,
                                sHost       := scParameter.fbstIp.stValue,
                                wPort       := scParameter.fbwPort.wValue,
                                eFrameType  := WagoAppPlcModbus.eMbFrameType.ETHERNET,
                                tTimeOut    := scParameter.fbtTimeOut.tValue,
                                utQuery     := fbJobFc6.utQuery,
                                xTrigger    := xTrigFc6,
                                utResponse  := fbJobFc6.utResponse);    												
END_IF;
(* Get Response *) 
IF usiState = 6 AND NOT xTrigFc6 AND fbJobFc6.xIsLocked AND NOT fbJobFc6.xJobDone THEN    
    usiState            := usiState + 1;
    ltMessungFc6        := fbTIMEFc6.Stop();
    metCheckOnError();
    fbJobFc6.metCallAfterResponse(fbMbClientUdp.xError,fbMbClientUdp.oStatus.uiID);
END_IF;
END_ACTION

PROPERTY proModBusErrorText : String(20)
GET
proModBusErrorText := TO_STRING(MAX(fbJobFc1.eError,fbJobFc2.eError,fbJobFc3.eError,fbJobFc4.eError,fbJobFc5.eError,fbJobFc6.eError,fbJobFc15.eError,fbJobFc16.eError));
END_GET
END_PROPERTY

PROPERTY proModBusEnabled : BOOL
GET
proModBusEnabled := scParameter.fbxEnable.xValue;
END_GET
END_PROPERTY

METHOD metITF_BMK
VAR_INPUT
	ITF_BMK_IN : CtaAppBmk.ITF_BMK;
END_VAR
ITF_BMK := ITF_BMK_IN;
END_METHOD

PROPERTY proITF_BMK : CtaAppBmk.ITF_BMK
GET
proITF_BMK := ITF_BMK;
END_GET
END_PROPERTY

ACTION actDelay:
(* Delay Read *)
tonDelayRead(	IN	:= xTrigDelayRead AND xTrigDelayWrite,
			 	PT 	:= scParameter.fbtDelayRead.proValue);
(* Delay Write *)
tonDelayWrite(	IN	:= xTrigDelayRead AND xTrigDelayWrite,
			 	PT 	:= scParameter.fbtDelayWrite.proValue);
				
(* Trig *)
xTrigDelayRead 	:= TRUE;
xTrigDelayWrite := TRUE;
END_ACTION

END_FUNCTION_BLOCK

// 30 Program Organization Units/CLIENT/SERIAL Client/fbMbSerialPortControll
FUNCTION_BLOCK fbMbSerialPortControll IMPLEMENTS ITF_MbPortControllSerial
VAR_INPUT
    I_Port                      :   WagoTypesCom.I_WagoSysComBase;
END_VAR
VAR
    fbMbClientSerial            : WagoAppPLCModbus.FbMbMasterSerial;
    bIdOfCourrentCall           : BYTE  := 1;
    bCountetCalls               : BYTE;
    fbConfigFile                : CtaSysConfig.fbConfigFile;
    scParameter                 : scSerialPortParameter;
    ayNodes                     : ARRAY[1..32] OF ITF_SERIAL_NODE;
    ayShowNodes                 : ARRAY[1..32] OF BOOL;
END_VAR

actConfig();

METHOD FINAL metSyncClient : BOOL
VAR_IN_OUT
    xAllJobsDone    : BOOL;
    bIdOfCall       : BYTE;
END_VAR
VAR_INPUT
    ITF_SERIAL_NODE : ITF_SERIAL_NODE;
END_VAR
IF bIdOfCall = 0 THEN
    IF bCountetCalls < 32 THEN
        bCountetCalls           := bCountetCalls + 1;
        bIdOfCall               := bCountetCalls;
        ayNodes[bIdOfCall]      := ITF_SERIAL_NODE;
        ayShowNodes[bIdOfCall]  := __QUERYINTERFACE(ITF_SERIAL_NODE,ITF_SERIAL_NODE);
    END_IF;   
END_IF;
IF bIdOfCourrentCall = 0 THEN
    bIdOfCourrentCall := 1;
END_IF;
IF bIdOfCall = bIdOfCourrentCall THEN
    IF xAllJobsDone THEN
        bIdOfCourrentCall := bIdOfCourrentCall + 1;
        IF bIdOfCourrentCall > bCountetCalls THEN
            bIdOfCourrentCall := 1;    
		END_IF
        metSyncClient := FALSE;
    ELSE
        metSyncClient := TRUE;
    END_IF;
END_IF;
END_METHOD

